// TIA Portal V20 export
FUNCTION_BLOCK "Sequence_1_TransferPnPLeft"   // FB32856, LAD
TITLE = Sequence
// Sequence template programmend in ladder logic
// stored: IsIECCheckEnabled true, MemoryReserve 100, Namespace Unit1.Em5, SetENOAutomatically true
   VAR_INPUT
      unitStatus { ExternalAccessible := 'False'; ExternalVisible := 'False'; ExternalWritable := 'False'} : "LAF_typeUnitStatus";
   END_VAR
   VAR
      instSequenceLADControl { ExternalAccessible := 'False'; ExternalVisible := 'False'; ExternalWritable := 'False'} : "LAF_ControlLadSequence";
      instSequenceLADStatus { ExternalAccessible := 'False'; ExternalVisible := 'False'; ExternalWritable := 'False'} : "LAF_StatusLadSequence";
      statTonTime { ExternalAccessible := 'False'; ExternalVisible := 'False'; ExternalWritable := 'False'} : Array[0..9999] of TON_TIME;
      NoDataCheck { S7_SetPoint := 'True'} : "LER_typePartData";
   END_VAR
   VAR_TEMP
      tempCustomerAction : Bool;   // Placeholder for possible actions
      tempDo_nothing_and_wait_for_init : Bool;   // Placeholder for doing nothing
      tempSafeStateCondition : Bool;   // Temp Condition for the equipment module to be in a safe state
   END_VAR
   VAR CONSTANT
      delayTime : Time := T#500ms;
      STEP_IDLE : DInt := 1;
      JOB_1_STEP_01 : DInt := 101;
      JOB_1_STEP_10 : DInt := 110;
      JOB_1_STEP_20 : DInt := 120;
      JOB_1_STEP_30 : DInt := 130;
      JOB_1_STEP_40 : DInt := 140;
      JOB_1_STEP_50 : DInt := 150;
      JOB_1_STEP_60 : DInt := 160;
      JOB_1_STEP_70 : DInt := 170;
      JOB_1_STEP_80 : DInt := 180;
      JOB_1_STEP_90 : DInt := 190;
      JOB_2_STEP_01 : DInt := 201;
      JOB_2_STEP_10 : DInt := 210;
      JOB_2_STEP_20 : DInt := 220;
      JOB_2_STEP_30 : DInt := 230;
      JOB_2_STEP_40 : DInt := 240;
      JOB_2_STEP_41 : DInt := 241;
      JOB_2_STEP_42 : DInt := 242;
      JOB_2_STEP_50 : DInt := 250;
      JOB_2_STEP_80 : DInt := 280;
      JOB_2_STEP_81 : DInt := 281;
      JOB_2_STEP_90 : DInt := 290;
      JOB_3_STEP_01 : DInt := 301;
      JOB_3_STEP_10 : DInt := 310;
      JOB_3_STEP_20 : DInt := 320;
      JOB_3_STEP_30 : DInt := 330;
      JOB_3_STEP_40 : DInt := 340;
      JOB_3_STEP_50 : DInt := 350;
      JOB_3_STEP_51 : DInt := 351;
      JOB_3_STEP_80 : DInt := 380;
      JOB_3_STEP_81 : DInt := 381;
      JOB_3_STEP_90 : DInt := 390;
      JOB_4_STEP_01 : DInt := 401;
      JOB_4_STEP_10 : DInt := 410;
      JOB_4_STEP_20 : DInt := 420;
      JOB_4_STEP_30 : DInt := 430;
      JOB_4_STEP_40 : DInt := 440;
      JOB_4_STEP_41 : DInt := 441;
      JOB_4_STEP_80 : DInt := 480;
      JOB_4_STEP_81 : DInt := 481;
      JOB_4_STEP_90 : DInt := 490;
      JOB_5_STEP_01 : DInt := 501;
      JOB_5_STEP_10 : DInt := 510;
      JOB_5_STEP_20 : DInt := 520;
      JOB_5_STEP_30 : DInt := 530;
      JOB_5_STEP_40 : DInt := 540;
      JOB_5_STEP_41 : DInt := 541;
      JOB_5_STEP_42 : DInt := 542;
      JOB_5_STEP_80 : DInt := 580;
      JOB_5_STEP_81 : DInt := 581;
      JOB_5_STEP_90 : DInt := 590;
      JOB_6_STEP_01 : DInt := 601;
      JOB_6_STEP_10 : DInt := 610;
      JOB_6_STEP_20 : DInt := 620;
      JOB_6_STEP_30 : DInt := 630;
      JOB_6_STEP_40 : DInt := 640;
      JOB_6_STEP_50 : DInt := 650;
      JOB_6_STEP_51 : DInt := 651;
      JOB_6_STEP_80 : DInt := 680;
      JOB_6_STEP_81 : DInt := 681;
      JOB_6_STEP_90 : DInt := 690;
      JOB_7_STEP_01 : DInt := 701;
      JOB_7_STEP_10 : DInt := 710;
      JOB_7_STEP_20 : DInt := 720;
      JOB_7_STEP_30 : DInt := 730;
      JOB_7_STEP_40 : DInt := 740;
      JOB_7_STEP_41 : DInt := 741;
      JOB_7_STEP_80 : DInt := 780;
      JOB_7_STEP_81 : DInt := 781;
      JOB_7_STEP_90 : DInt := 790;
      JOB_9_STEP_01 : DInt := 901;
      JOB_9_STEP_10 : DInt := 910;
      JOB_9_STEP_20 : DInt := 920;
      JOB_9_STEP_30 : DInt := 930;
      JOB_9_STEP_40 : DInt := 940;
      JOB_9_STEP_50 : DInt := 950;
      JOB_9_STEP_51 : DInt := 951;
      JOB_9_STEP_80 : DInt := 980;
      JOB_9_STEP_81 : DInt := 981;
      JOB_9_STEP_82 : DInt := 982;
      JOB_9_STEP_90 : DInt := 990;
      STEP_IMMEDIATE_STOP : DInt := 9001;   // Step executed when an immediate stop command is triggered for the sequence (i.e. when unit is in state aborting)
   END_VAR
   VAR_TEMP   // added for the SCL form of the ladder/FBD networks
      _w1 : Bool;
      _w2 : Bool;
      _w3 : Bool;
      _w4 : Bool;
      _w5 : Bool;
      _w6 : Bool;
      _w7 : Bool;
   END_VAR
BEGIN

REGION Network 1: BLOCK INFO HEADER
   // (company) / (C) Copyright (year)
   // ---------------------------------------------------------------------------------
   // Title:                             (Title of this block)
   // Comment/Function: (that is implemented in the block)
   // Library/Family:           (that the source is dedicated to)
   // Author:                        (department / person in charge / contact)
   // Target System:          (test system with FW version)
   // Engineering:              TIA Portal (SW version)
   // Restrictions:               (OB types, etc.)
   // Requirements:           (hardware, technological package, etc.)
   // ---------------------------------------------------------------------------------
   // Change log table:
   // Version          | Date             | Signature      | Expert in charge  | Changes applied ------------------------|----------------------|-------------------------|--------------------------------|-----------------------
   // 001.000.000 | yyyy-mm-dd | 0x00000000 | (name of expert) | First released version
END_REGION

REGION Network 2: DESCRIPTION
   // This is a template block provided by the Automation Framework. It can be used to create an own project.
   // The Block Info Header is prepared to put in your own data.
   // Description of the block could be added here and the docu created by Code2Docu.
END_REGION

REGION Network 3: ********************* CONTROL *************************
END_REGION

REGION Network 4: Sequence Control ("Enter your Sequins number here")
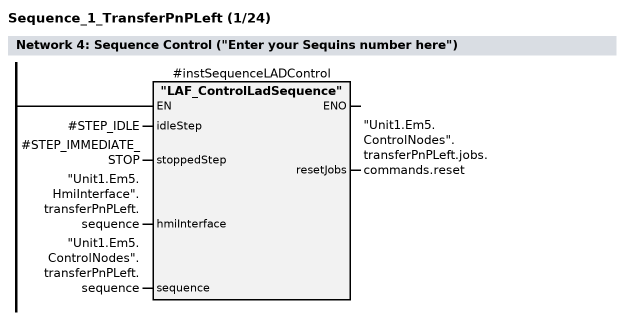
   RUNG wire#powerrail
      #instSequenceLADControl(idleStep := #STEP_IDLE, stoppedStep := #STEP_IMMEDIATE_STOP, hmiInterface := "Unit1.Em5.HmiInterface".transferPnPLeft.sequence, sequence := "Unit1.Em5.ControlNodes".transferPnPLeft.sequence, resetJobs => "Unit1.Em5.ControlNodes".transferPnPLeft.jobs.commands.reset)
   END_RUNG
   // the same network as SCL:
   #instSequenceLADControl(idleStep := #STEP_IDLE,   // "LAF_ControlLadSequence"
                           stoppedStep := #STEP_IMMEDIATE_STOP,
                           hmiInterface := "Unit1.Em5.HmiInterface".transferPnPLeft.sequence,
                           sequence := "Unit1.Em5.ControlNodes".transferPnPLeft.sequence,
                           resetJobs => "Unit1.Em5.ControlNodes".transferPnPLeft.jobs.commands.reset);
END_REGION

REGION Network 5: Step IDLE
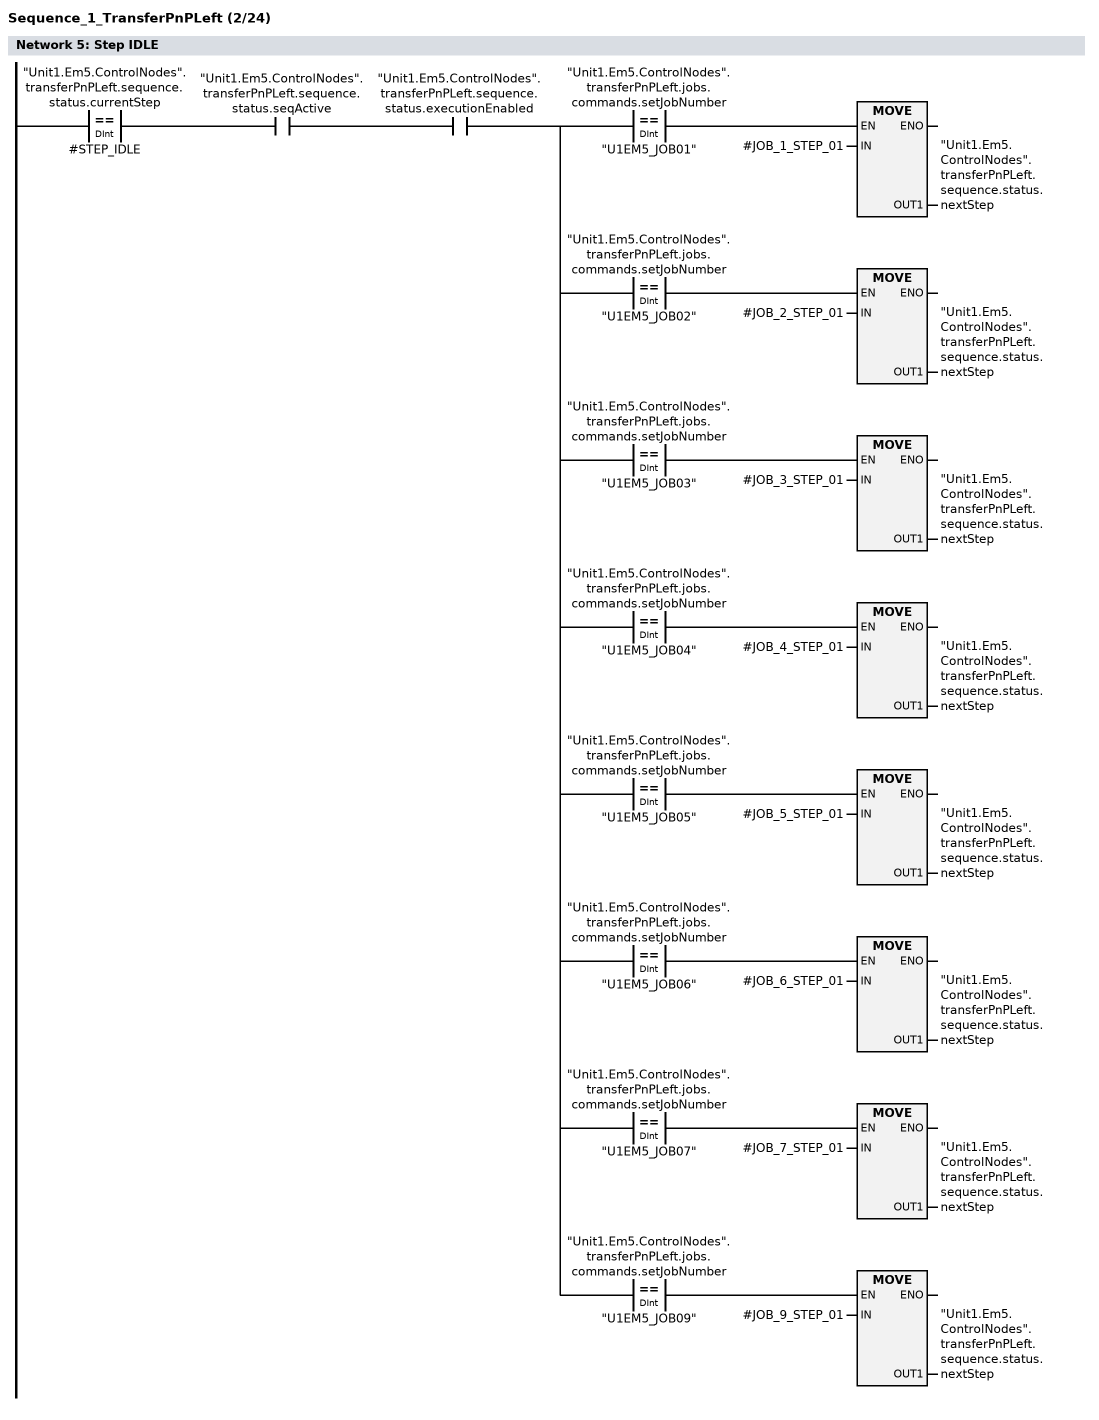
   RUNG wire#powerrail
      { S7_Templates := "SrcType := DInt" } EQ_Contact(in1 := "Unit1.Em5.ControlNodes".transferPnPLeft.sequence.status.currentStep, in2 := #STEP_IDLE)
      Contact( "Unit1.Em5.ControlNodes".transferPnPLeft.sequence.status.seqActive )
      Contact( "Unit1.Em5.ControlNodes".transferPnPLeft.sequence.status.executionEnabled )
      wire#w1
      { S7_Templates := "SrcType := DInt" } EQ_Contact(in1 := "Unit1.Em5.ControlNodes".transferPnPLeft.jobs.commands.setJobNumber, in2 := "U1EM5_JOB01")
      Move(in := #JOB_1_STEP_01, out1 => "Unit1.Em5.ControlNodes".transferPnPLeft.sequence.status.nextStep)
   END_RUNG
   RUNG wire#w1
      { S7_Templates := "SrcType := DInt" } EQ_Contact(in1 := "Unit1.Em5.ControlNodes".transferPnPLeft.jobs.commands.setJobNumber, in2 := "U1EM5_JOB02")
      Move(in := #JOB_2_STEP_01, out1 => "Unit1.Em5.ControlNodes".transferPnPLeft.sequence.status.nextStep)
   END_RUNG
   RUNG wire#w1
      { S7_Templates := "SrcType := DInt" } EQ_Contact(in1 := "Unit1.Em5.ControlNodes".transferPnPLeft.jobs.commands.setJobNumber, in2 := "U1EM5_JOB03")
      Move(in := #JOB_3_STEP_01, out1 => "Unit1.Em5.ControlNodes".transferPnPLeft.sequence.status.nextStep)
   END_RUNG
   RUNG wire#w1
      { S7_Templates := "SrcType := DInt" } EQ_Contact(in1 := "Unit1.Em5.ControlNodes".transferPnPLeft.jobs.commands.setJobNumber, in2 := "U1EM5_JOB04")
      Move(in := #JOB_4_STEP_01, out1 => "Unit1.Em5.ControlNodes".transferPnPLeft.sequence.status.nextStep)
   END_RUNG
   RUNG wire#w1
      { S7_Templates := "SrcType := DInt" } EQ_Contact(in1 := "Unit1.Em5.ControlNodes".transferPnPLeft.jobs.commands.setJobNumber, in2 := "U1EM5_JOB05")
      Move(in := #JOB_5_STEP_01, out1 => "Unit1.Em5.ControlNodes".transferPnPLeft.sequence.status.nextStep)
   END_RUNG
   RUNG wire#w1
      { S7_Templates := "SrcType := DInt" } EQ_Contact(in1 := "Unit1.Em5.ControlNodes".transferPnPLeft.jobs.commands.setJobNumber, in2 := "U1EM5_JOB06")
      Move(in := #JOB_6_STEP_01, out1 => "Unit1.Em5.ControlNodes".transferPnPLeft.sequence.status.nextStep)
   END_RUNG
   RUNG wire#w1
      { S7_Templates := "SrcType := DInt" } EQ_Contact(in1 := "Unit1.Em5.ControlNodes".transferPnPLeft.jobs.commands.setJobNumber, in2 := "U1EM5_JOB07")
      Move(in := #JOB_7_STEP_01, out1 => "Unit1.Em5.ControlNodes".transferPnPLeft.sequence.status.nextStep)
   END_RUNG
   RUNG wire#w1
      { S7_Templates := "SrcType := DInt" } EQ_Contact(in1 := "Unit1.Em5.ControlNodes".transferPnPLeft.jobs.commands.setJobNumber, in2 := "U1EM5_JOB09")
      Move(in := #JOB_9_STEP_01, out1 => "Unit1.Em5.ControlNodes".transferPnPLeft.sequence.status.nextStep)
   END_RUNG
   // the same network as SCL:
   #_w1 := ("Unit1.Em5.ControlNodes".transferPnPLeft.sequence.status.currentStep = #STEP_IDLE) AND "Unit1.Em5.ControlNodes".transferPnPLeft.sequence.status.seqActive AND "Unit1.Em5.ControlNodes".transferPnPLeft.sequence.status.executionEnabled;
   IF #_w1 AND ("Unit1.Em5.ControlNodes".transferPnPLeft.jobs.commands.setJobNumber = "U1EM5_JOB01") THEN
       "Unit1.Em5.ControlNodes".transferPnPLeft.sequence.status.nextStep := #JOB_1_STEP_01;
   END_IF;
   IF #_w1 AND ("Unit1.Em5.ControlNodes".transferPnPLeft.jobs.commands.setJobNumber = "U1EM5_JOB02") THEN
       "Unit1.Em5.ControlNodes".transferPnPLeft.sequence.status.nextStep := #JOB_2_STEP_01;
   END_IF;
   IF #_w1 AND ("Unit1.Em5.ControlNodes".transferPnPLeft.jobs.commands.setJobNumber = "U1EM5_JOB03") THEN
       "Unit1.Em5.ControlNodes".transferPnPLeft.sequence.status.nextStep := #JOB_3_STEP_01;
   END_IF;
   IF #_w1 AND ("Unit1.Em5.ControlNodes".transferPnPLeft.jobs.commands.setJobNumber = "U1EM5_JOB04") THEN
       "Unit1.Em5.ControlNodes".transferPnPLeft.sequence.status.nextStep := #JOB_4_STEP_01;
   END_IF;
   IF #_w1 AND ("Unit1.Em5.ControlNodes".transferPnPLeft.jobs.commands.setJobNumber = "U1EM5_JOB05") THEN
       "Unit1.Em5.ControlNodes".transferPnPLeft.sequence.status.nextStep := #JOB_5_STEP_01;
   END_IF;
   IF #_w1 AND ("Unit1.Em5.ControlNodes".transferPnPLeft.jobs.commands.setJobNumber = "U1EM5_JOB06") THEN
       "Unit1.Em5.ControlNodes".transferPnPLeft.sequence.status.nextStep := #JOB_6_STEP_01;
   END_IF;
   IF #_w1 AND ("Unit1.Em5.ControlNodes".transferPnPLeft.jobs.commands.setJobNumber = "U1EM5_JOB07") THEN
       "Unit1.Em5.ControlNodes".transferPnPLeft.sequence.status.nextStep := #JOB_7_STEP_01;
   END_IF;
   IF #_w1 AND ("Unit1.Em5.ControlNodes".transferPnPLeft.jobs.commands.setJobNumber = "U1EM5_JOB09") THEN
       "Unit1.Em5.ControlNodes".transferPnPLeft.sequence.status.nextStep := #JOB_9_STEP_01;
   END_IF;
END_REGION

REGION Network 6: *************** JOB[1] EM HOMING ************************
END_REGION

REGION Network 7: Step[101] : JOB[1] Condition
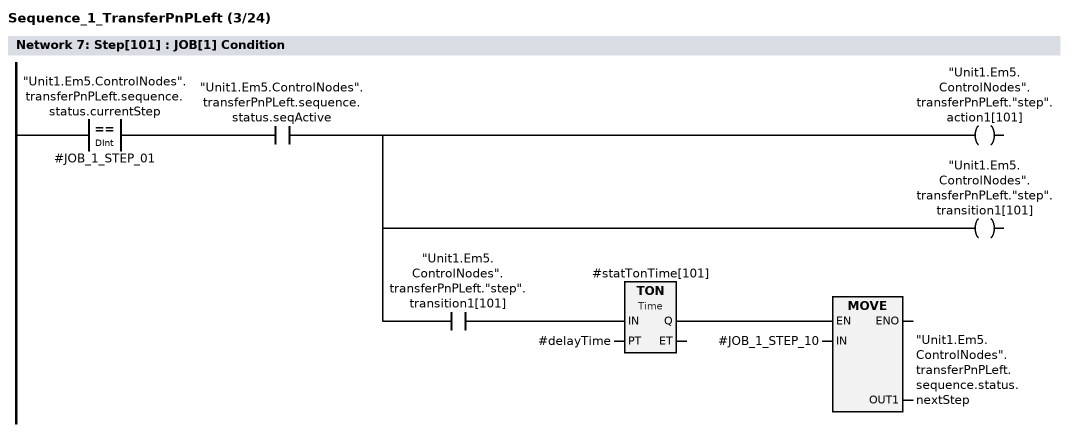
   RUNG wire#powerrail
      { S7_Templates := "SrcType := DInt" } EQ_Contact(in1 := "Unit1.Em5.ControlNodes".transferPnPLeft.sequence.status.currentStep, in2 := #JOB_1_STEP_01)
      Contact( "Unit1.Em5.ControlNodes".transferPnPLeft.sequence.status.seqActive )
      wire#w1
      Coil( "Unit1.Em5.ControlNodes".transferPnPLeft."step".action1[101] )
   END_RUNG
   RUNG wire#w1
      Coil( "Unit1.Em5.ControlNodes".transferPnPLeft."step".transition1[101] )
   END_RUNG
   RUNG wire#w1
      Contact( "Unit1.Em5.ControlNodes".transferPnPLeft."step".transition1[101] )
      { S7_Templates := "time_type := Time" } #statTonTime[101].TON(pt := #delayTime, et =>)
      Move(in := #JOB_1_STEP_10, out1 => "Unit1.Em5.ControlNodes".transferPnPLeft.sequence.status.nextStep)
   END_RUNG
   // the same network as SCL:
   "Unit1.Em5.ControlNodes".transferPnPLeft."step".action1[101] := ("Unit1.Em5.ControlNodes".transferPnPLeft.sequence.status.currentStep = #JOB_1_STEP_01) AND "Unit1.Em5.ControlNodes".transferPnPLeft.sequence.status.seqActive;
   "Unit1.Em5.ControlNodes".transferPnPLeft."step".transition1[101] := ("Unit1.Em5.ControlNodes".transferPnPLeft.sequence.status.currentStep = #JOB_1_STEP_01) AND "Unit1.Em5.ControlNodes".transferPnPLeft.sequence.status.seqActive;
   #statTonTime[101].TON(IN := ("Unit1.Em5.ControlNodes".transferPnPLeft.sequence.status.currentStep = #JOB_1_STEP_01) AND "Unit1.Em5.ControlNodes".transferPnPLeft.sequence.status.seqActive AND "Unit1.Em5.ControlNodes".transferPnPLeft."step".transition1[101],
                         PT := #delayTime);
   IF #statTonTime[101].Q THEN
       "Unit1.Em5.ControlNodes".transferPnPLeft.sequence.status.nextStep := #JOB_1_STEP_10;
   END_IF;
END_REGION

REGION Network 8: Step[110] : Transfer PP Left Clamp Open
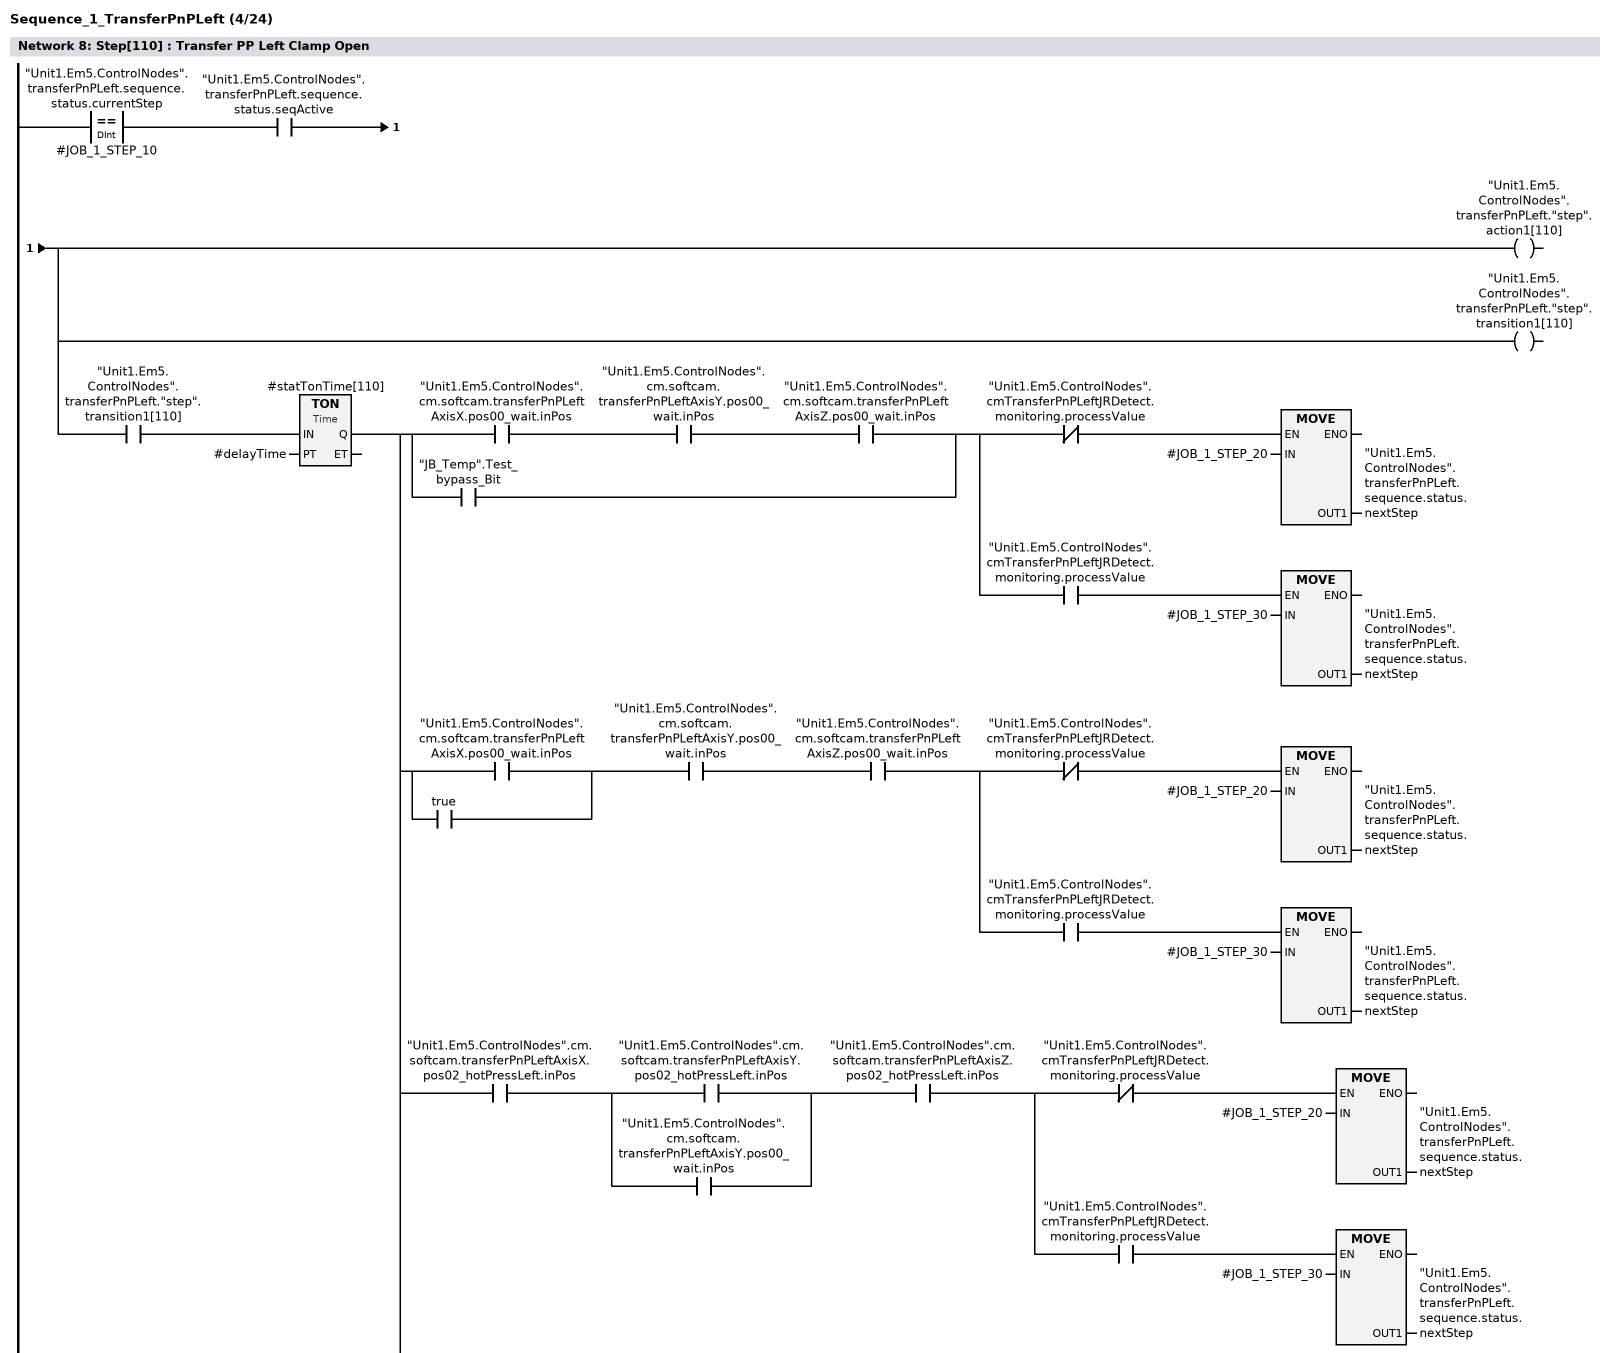
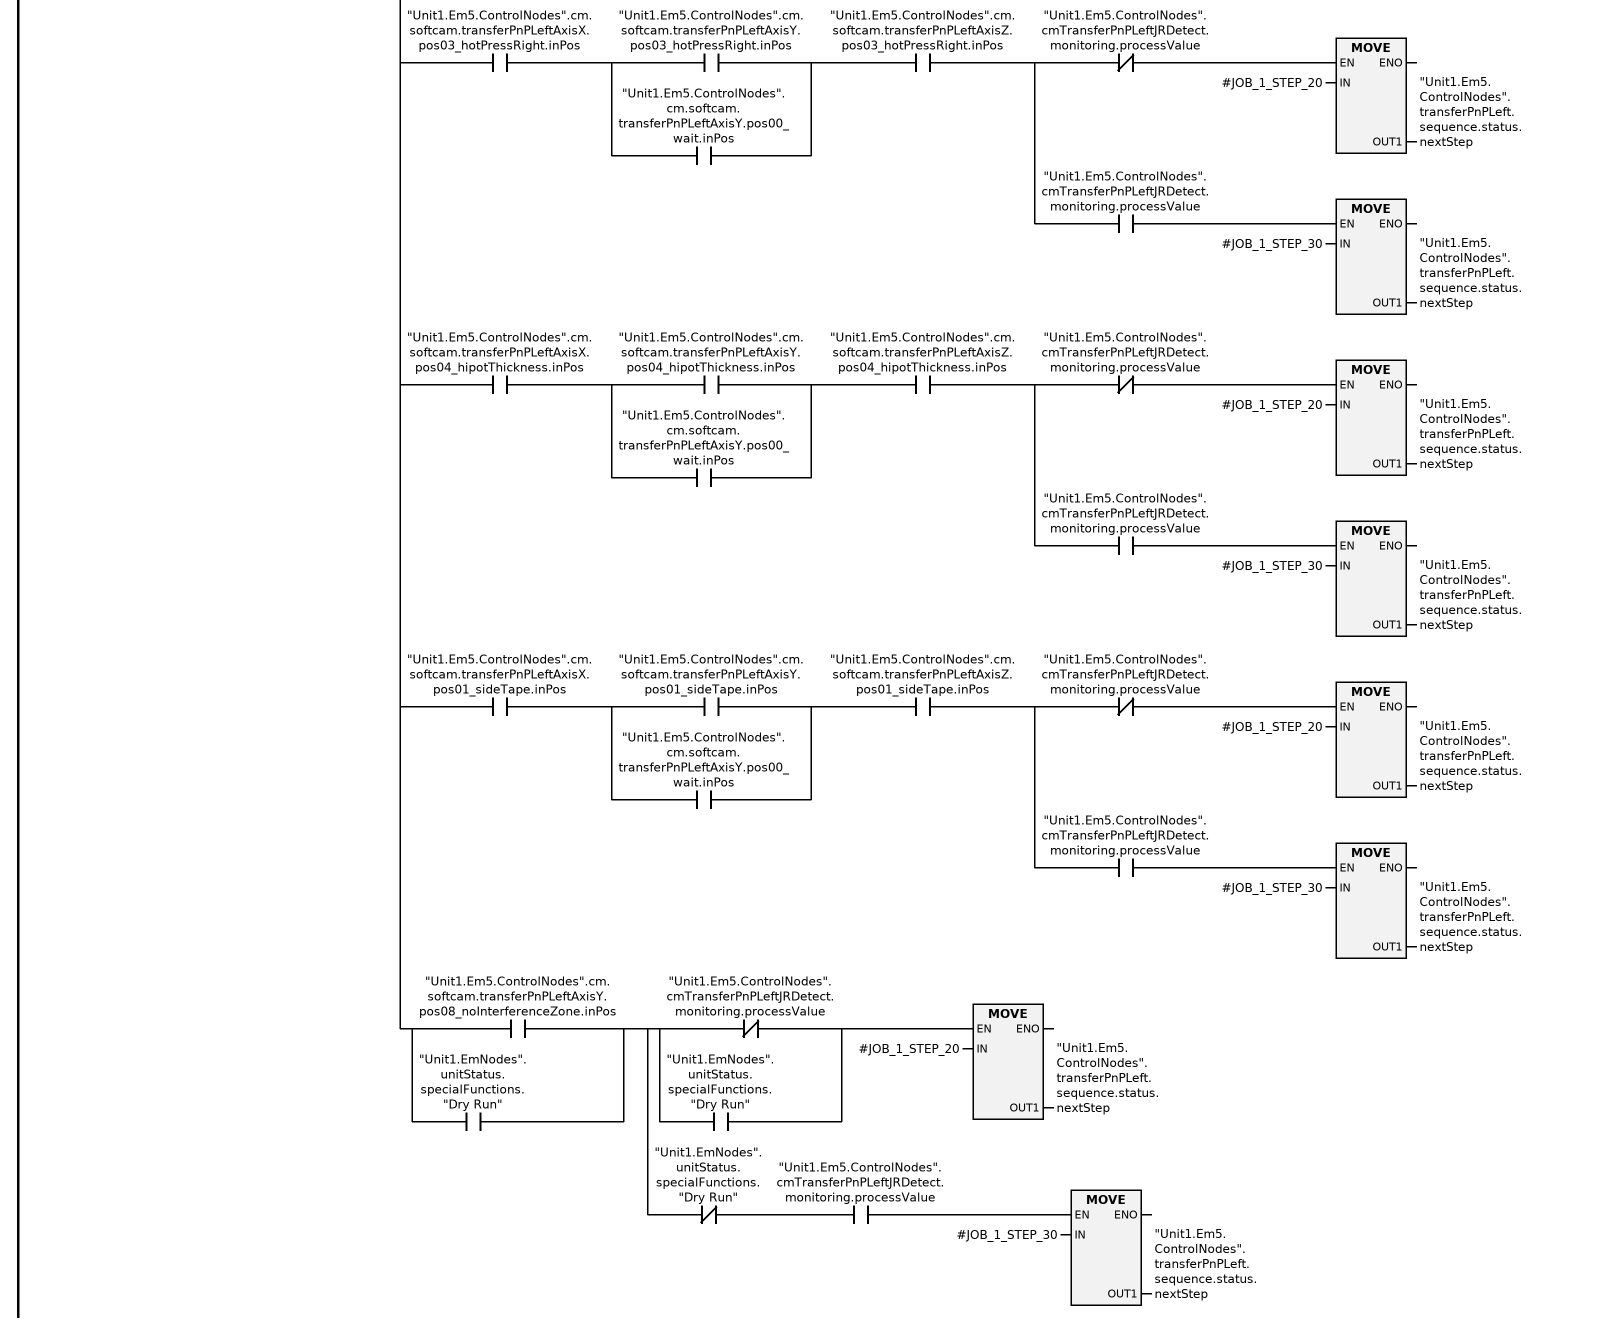
   RUNG wire#powerrail
      { S7_Templates := "SrcType := DInt" } EQ_Contact(in1 := "Unit1.Em5.ControlNodes".transferPnPLeft.sequence.status.currentStep, in2 := #JOB_1_STEP_10)
      Contact( "Unit1.Em5.ControlNodes".transferPnPLeft.sequence.status.seqActive )
      wire#w1
      Coil( "Unit1.Em5.ControlNodes".transferPnPLeft."step".action1[110] )
   END_RUNG
   RUNG wire#w1
      Coil( "Unit1.Em5.ControlNodes".transferPnPLeft."step".transition1[110] )
   END_RUNG
   RUNG wire#w1
      Contact( "Unit1.Em5.ControlNodes".transferPnPLeft."step".transition1[110] )
      { S7_Templates := "time_type := Time" } #statTonTime[110].TON(pt := #delayTime, et =>)
      wire#w2
      Contact( "Unit1.Em5.ControlNodes".cm.softcam.transferPnPLeftAxisX.pos00_wait.inPos )
      Contact( "Unit1.Em5.ControlNodes".cm.softcam.transferPnPLeftAxisY.pos00_wait.inPos )
      Contact( "Unit1.Em5.ControlNodes".cm.softcam.transferPnPLeftAxisZ.pos00_wait.inPos )
      wire#w3
      I_Contact( "Unit1.Em5.ControlNodes".cmTransferPnPLeftJRDetect.monitoring.processValue )
      Move(in := #JOB_1_STEP_20, out1 => "Unit1.Em5.ControlNodes".transferPnPLeft.sequence.status.nextStep)
   END_RUNG
   RUNG wire#w2
      Contact( "JB_Temp".Test_bypass_Bit )
   END_RUNG wire#w3
   RUNG wire#w3
      Contact( "Unit1.Em5.ControlNodes".cmTransferPnPLeftJRDetect.monitoring.processValue )
      Move(in := #JOB_1_STEP_30, out1 => "Unit1.Em5.ControlNodes".transferPnPLeft.sequence.status.nextStep)
   END_RUNG
   RUNG wire#w2
      Contact( "Unit1.Em5.ControlNodes".cm.softcam.transferPnPLeftAxisX.pos00_wait.inPos )
      wire#w4
      Contact( "Unit1.Em5.ControlNodes".cm.softcam.transferPnPLeftAxisY.pos00_wait.inPos )
      Contact( "Unit1.Em5.ControlNodes".cm.softcam.transferPnPLeftAxisZ.pos00_wait.inPos )
      wire#w5
      I_Contact( "Unit1.Em5.ControlNodes".cmTransferPnPLeftJRDetect.monitoring.processValue )
      Move(in := #JOB_1_STEP_20, out1 => "Unit1.Em5.ControlNodes".transferPnPLeft.sequence.status.nextStep)
   END_RUNG
   RUNG wire#w2
      Contact( true )
   END_RUNG wire#w4
   RUNG wire#w5
      Contact( "Unit1.Em5.ControlNodes".cmTransferPnPLeftJRDetect.monitoring.processValue )
      Move(in := #JOB_1_STEP_30, out1 => "Unit1.Em5.ControlNodes".transferPnPLeft.sequence.status.nextStep)
   END_RUNG
   RUNG wire#w2
      Contact( "Unit1.Em5.ControlNodes".cm.softcam.transferPnPLeftAxisX.pos02_hotPressLeft.inPos )
      wire#w6
      Contact( "Unit1.Em5.ControlNodes".cm.softcam.transferPnPLeftAxisY.pos02_hotPressLeft.inPos )
      wire#w7
      Contact( "Unit1.Em5.ControlNodes".cm.softcam.transferPnPLeftAxisZ.pos02_hotPressLeft.inPos )
      wire#w8
      I_Contact( "Unit1.Em5.ControlNodes".cmTransferPnPLeftJRDetect.monitoring.processValue )
      Move(in := #JOB_1_STEP_20, out1 => "Unit1.Em5.ControlNodes".transferPnPLeft.sequence.status.nextStep)
   END_RUNG
   RUNG wire#w6
      Contact( "Unit1.Em5.ControlNodes".cm.softcam.transferPnPLeftAxisY.pos00_wait.inPos )
   END_RUNG wire#w7
   RUNG wire#w8
      Contact( "Unit1.Em5.ControlNodes".cmTransferPnPLeftJRDetect.monitoring.processValue )
      Move(in := #JOB_1_STEP_30, out1 => "Unit1.Em5.ControlNodes".transferPnPLeft.sequence.status.nextStep)
   END_RUNG
   RUNG wire#w2
      Contact( "Unit1.Em5.ControlNodes".cm.softcam.transferPnPLeftAxisX.pos03_hotPressRight.inPos )
      wire#w9
      Contact( "Unit1.Em5.ControlNodes".cm.softcam.transferPnPLeftAxisY.pos03_hotPressRight.inPos )
      wire#w10
      Contact( "Unit1.Em5.ControlNodes".cm.softcam.transferPnPLeftAxisZ.pos03_hotPressRight.inPos )
      wire#w11
      I_Contact( "Unit1.Em5.ControlNodes".cmTransferPnPLeftJRDetect.monitoring.processValue )
      Move(in := #JOB_1_STEP_20, out1 => "Unit1.Em5.ControlNodes".transferPnPLeft.sequence.status.nextStep)
   END_RUNG
   RUNG wire#w9
      Contact( "Unit1.Em5.ControlNodes".cm.softcam.transferPnPLeftAxisY.pos00_wait.inPos )
   END_RUNG wire#w10
   RUNG wire#w11
      Contact( "Unit1.Em5.ControlNodes".cmTransferPnPLeftJRDetect.monitoring.processValue )
      Move(in := #JOB_1_STEP_30, out1 => "Unit1.Em5.ControlNodes".transferPnPLeft.sequence.status.nextStep)
   END_RUNG
   RUNG wire#w2
      Contact( "Unit1.Em5.ControlNodes".cm.softcam.transferPnPLeftAxisX.pos04_hipotThickness.inPos )
      wire#w12
      Contact( "Unit1.Em5.ControlNodes".cm.softcam.transferPnPLeftAxisY.pos04_hipotThickness.inPos )
      wire#w13
      Contact( "Unit1.Em5.ControlNodes".cm.softcam.transferPnPLeftAxisZ.pos04_hipotThickness.inPos )
      wire#w14
      I_Contact( "Unit1.Em5.ControlNodes".cmTransferPnPLeftJRDetect.monitoring.processValue )
      Move(in := #JOB_1_STEP_20, out1 => "Unit1.Em5.ControlNodes".transferPnPLeft.sequence.status.nextStep)
   END_RUNG
   RUNG wire#w12
      Contact( "Unit1.Em5.ControlNodes".cm.softcam.transferPnPLeftAxisY.pos00_wait.inPos )
   END_RUNG wire#w13
   RUNG wire#w14
      Contact( "Unit1.Em5.ControlNodes".cmTransferPnPLeftJRDetect.monitoring.processValue )
      Move(in := #JOB_1_STEP_30, out1 => "Unit1.Em5.ControlNodes".transferPnPLeft.sequence.status.nextStep)
   END_RUNG
   RUNG wire#w2
      Contact( "Unit1.Em5.ControlNodes".cm.softcam.transferPnPLeftAxisX.pos01_sideTape.inPos )
      wire#w15
      Contact( "Unit1.Em5.ControlNodes".cm.softcam.transferPnPLeftAxisY.pos01_sideTape.inPos )
      wire#w16
      Contact( "Unit1.Em5.ControlNodes".cm.softcam.transferPnPLeftAxisZ.pos01_sideTape.inPos )
      wire#w17
      I_Contact( "Unit1.Em5.ControlNodes".cmTransferPnPLeftJRDetect.monitoring.processValue )
      Move(in := #JOB_1_STEP_20, out1 => "Unit1.Em5.ControlNodes".transferPnPLeft.sequence.status.nextStep)
   END_RUNG
   RUNG wire#w15
      Contact( "Unit1.Em5.ControlNodes".cm.softcam.transferPnPLeftAxisY.pos00_wait.inPos )
   END_RUNG wire#w16
   RUNG wire#w17
      Contact( "Unit1.Em5.ControlNodes".cmTransferPnPLeftJRDetect.monitoring.processValue )
      Move(in := #JOB_1_STEP_30, out1 => "Unit1.Em5.ControlNodes".transferPnPLeft.sequence.status.nextStep)
   END_RUNG
   RUNG wire#w2
      Contact( "Unit1.Em5.ControlNodes".cm.softcam.transferPnPLeftAxisY.pos08_noInterferenceZone.inPos )
      wire#w18
      I_Contact( "Unit1.Em5.ControlNodes".cmTransferPnPLeftJRDetect.monitoring.processValue )
      wire#w19
      Move(in := #JOB_1_STEP_20, out1 => "Unit1.Em5.ControlNodes".transferPnPLeft.sequence.status.nextStep)
   END_RUNG
   RUNG wire#w2
      Contact( "Unit1.EmNodes".unitStatus.specialFunctions."Dry Run" )
   END_RUNG wire#w18
   RUNG wire#w18
      Contact( "Unit1.EmNodes".unitStatus.specialFunctions."Dry Run" )
   END_RUNG wire#w19
   RUNG wire#w18
      I_Contact( "Unit1.EmNodes".unitStatus.specialFunctions."Dry Run" )
      Contact( "Unit1.Em5.ControlNodes".cmTransferPnPLeftJRDetect.monitoring.processValue )
      Move(in := #JOB_1_STEP_30, out1 => "Unit1.Em5.ControlNodes".transferPnPLeft.sequence.status.nextStep)
   END_RUNG
   // the same network as SCL:
   "Unit1.Em5.ControlNodes".transferPnPLeft."step".action1[110] := ("Unit1.Em5.ControlNodes".transferPnPLeft.sequence.status.currentStep = #JOB_1_STEP_10) AND "Unit1.Em5.ControlNodes".transferPnPLeft.sequence.status.seqActive;
   "Unit1.Em5.ControlNodes".transferPnPLeft."step".transition1[110] := ("Unit1.Em5.ControlNodes".transferPnPLeft.sequence.status.currentStep = #JOB_1_STEP_10) AND "Unit1.Em5.ControlNodes".transferPnPLeft.sequence.status.seqActive;
   #statTonTime[110].TON(IN := ("Unit1.Em5.ControlNodes".transferPnPLeft.sequence.status.currentStep = #JOB_1_STEP_10) AND "Unit1.Em5.ControlNodes".transferPnPLeft.sequence.status.seqActive AND "Unit1.Em5.ControlNodes".transferPnPLeft."step".transition1[110],
                         PT := #delayTime);
   #_w1 := #statTonTime[110].Q AND (("Unit1.Em5.ControlNodes".cm.softcam.transferPnPLeftAxisX.pos00_wait.inPos AND "Unit1.Em5.ControlNodes".cm.softcam.transferPnPLeftAxisY.pos00_wait.inPos AND "Unit1.Em5.ControlNodes".cm.softcam.transferPnPLeftAxisZ.pos00_wait.inPos) OR "JB_Temp".Test_bypass_Bit);
   IF #_w1 AND NOT "Unit1.Em5.ControlNodes".cmTransferPnPLeftJRDetect.monitoring.processValue THEN
       "Unit1.Em5.ControlNodes".transferPnPLeft.sequence.status.nextStep := #JOB_1_STEP_20;
   END_IF;
   IF #_w1 AND "Unit1.Em5.ControlNodes".cmTransferPnPLeftJRDetect.monitoring.processValue THEN
       "Unit1.Em5.ControlNodes".transferPnPLeft.sequence.status.nextStep := #JOB_1_STEP_30;
   END_IF;
   #_w2 := #statTonTime[110].Q AND ("Unit1.Em5.ControlNodes".cm.softcam.transferPnPLeftAxisX.pos00_wait.inPos OR true) AND "Unit1.Em5.ControlNodes".cm.softcam.transferPnPLeftAxisY.pos00_wait.inPos AND "Unit1.Em5.ControlNodes".cm.softcam.transferPnPLeftAxisZ.pos00_wait.inPos;
   IF #_w2 AND NOT "Unit1.Em5.ControlNodes".cmTransferPnPLeftJRDetect.monitoring.processValue THEN
       "Unit1.Em5.ControlNodes".transferPnPLeft.sequence.status.nextStep := #JOB_1_STEP_20;
   END_IF;
   IF #_w2 AND "Unit1.Em5.ControlNodes".cmTransferPnPLeftJRDetect.monitoring.processValue THEN
       "Unit1.Em5.ControlNodes".transferPnPLeft.sequence.status.nextStep := #JOB_1_STEP_30;
   END_IF;
   #_w3 := #statTonTime[110].Q AND "Unit1.Em5.ControlNodes".cm.softcam.transferPnPLeftAxisX.pos02_hotPressLeft.inPos AND ("Unit1.Em5.ControlNodes".cm.softcam.transferPnPLeftAxisY.pos02_hotPressLeft.inPos OR "Unit1.Em5.ControlNodes".cm.softcam.transferPnPLeftAxisY.pos00_wait.inPos) AND "Unit1.Em5.ControlNodes".cm.softcam.transferPnPLeftAxisZ.pos02_hotPressLeft.inPos;
   IF #_w3 AND NOT "Unit1.Em5.ControlNodes".cmTransferPnPLeftJRDetect.monitoring.processValue THEN
       "Unit1.Em5.ControlNodes".transferPnPLeft.sequence.status.nextStep := #JOB_1_STEP_20;
   END_IF;
   IF #_w3 AND "Unit1.Em5.ControlNodes".cmTransferPnPLeftJRDetect.monitoring.processValue THEN
       "Unit1.Em5.ControlNodes".transferPnPLeft.sequence.status.nextStep := #JOB_1_STEP_30;
   END_IF;
   #_w4 := #statTonTime[110].Q AND "Unit1.Em5.ControlNodes".cm.softcam.transferPnPLeftAxisX.pos03_hotPressRight.inPos AND ("Unit1.Em5.ControlNodes".cm.softcam.transferPnPLeftAxisY.pos03_hotPressRight.inPos OR "Unit1.Em5.ControlNodes".cm.softcam.transferPnPLeftAxisY.pos00_wait.inPos) AND "Unit1.Em5.ControlNodes".cm.softcam.transferPnPLeftAxisZ.pos03_hotPressRight.inPos;
   IF #_w4 AND NOT "Unit1.Em5.ControlNodes".cmTransferPnPLeftJRDetect.monitoring.processValue THEN
       "Unit1.Em5.ControlNodes".transferPnPLeft.sequence.status.nextStep := #JOB_1_STEP_20;
   END_IF;
   IF #_w4 AND "Unit1.Em5.ControlNodes".cmTransferPnPLeftJRDetect.monitoring.processValue THEN
       "Unit1.Em5.ControlNodes".transferPnPLeft.sequence.status.nextStep := #JOB_1_STEP_30;
   END_IF;
   #_w5 := #statTonTime[110].Q AND "Unit1.Em5.ControlNodes".cm.softcam.transferPnPLeftAxisX.pos04_hipotThickness.inPos AND ("Unit1.Em5.ControlNodes".cm.softcam.transferPnPLeftAxisY.pos04_hipotThickness.inPos OR "Unit1.Em5.ControlNodes".cm.softcam.transferPnPLeftAxisY.pos00_wait.inPos) AND "Unit1.Em5.ControlNodes".cm.softcam.transferPnPLeftAxisZ.pos04_hipotThickness.inPos;
   IF #_w5 AND NOT "Unit1.Em5.ControlNodes".cmTransferPnPLeftJRDetect.monitoring.processValue THEN
       "Unit1.Em5.ControlNodes".transferPnPLeft.sequence.status.nextStep := #JOB_1_STEP_20;
   END_IF;
   IF #_w5 AND "Unit1.Em5.ControlNodes".cmTransferPnPLeftJRDetect.monitoring.processValue THEN
       "Unit1.Em5.ControlNodes".transferPnPLeft.sequence.status.nextStep := #JOB_1_STEP_30;
   END_IF;
   #_w6 := #statTonTime[110].Q AND "Unit1.Em5.ControlNodes".cm.softcam.transferPnPLeftAxisX.pos01_sideTape.inPos AND ("Unit1.Em5.ControlNodes".cm.softcam.transferPnPLeftAxisY.pos01_sideTape.inPos OR "Unit1.Em5.ControlNodes".cm.softcam.transferPnPLeftAxisY.pos00_wait.inPos) AND "Unit1.Em5.ControlNodes".cm.softcam.transferPnPLeftAxisZ.pos01_sideTape.inPos;
   IF #_w6 AND NOT "Unit1.Em5.ControlNodes".cmTransferPnPLeftJRDetect.monitoring.processValue THEN
       "Unit1.Em5.ControlNodes".transferPnPLeft.sequence.status.nextStep := #JOB_1_STEP_20;
   END_IF;
   IF #_w6 AND "Unit1.Em5.ControlNodes".cmTransferPnPLeftJRDetect.monitoring.processValue THEN
       "Unit1.Em5.ControlNodes".transferPnPLeft.sequence.status.nextStep := #JOB_1_STEP_30;
   END_IF;
   #_w7 := #statTonTime[110].Q AND ("Unit1.Em5.ControlNodes".cm.softcam.transferPnPLeftAxisY.pos08_noInterferenceZone.inPos OR "Unit1.EmNodes".unitStatus.specialFunctions."Dry Run");
   IF #_w7 AND (NOT "Unit1.Em5.ControlNodes".cmTransferPnPLeftJRDetect.monitoring.processValue OR "Unit1.EmNodes".unitStatus.specialFunctions."Dry Run") THEN
       "Unit1.Em5.ControlNodes".transferPnPLeft.sequence.status.nextStep := #JOB_1_STEP_20;
   END_IF;
   IF #_w7 AND NOT "Unit1.EmNodes".unitStatus.specialFunctions."Dry Run" AND "Unit1.Em5.ControlNodes".cmTransferPnPLeftJRDetect.monitoring.processValue THEN
       "Unit1.Em5.ControlNodes".transferPnPLeft.sequence.status.nextStep := #JOB_1_STEP_30;
   END_IF;
END_REGION

REGION Network 9: Step[120] : Transfer PP Left Clamp Open
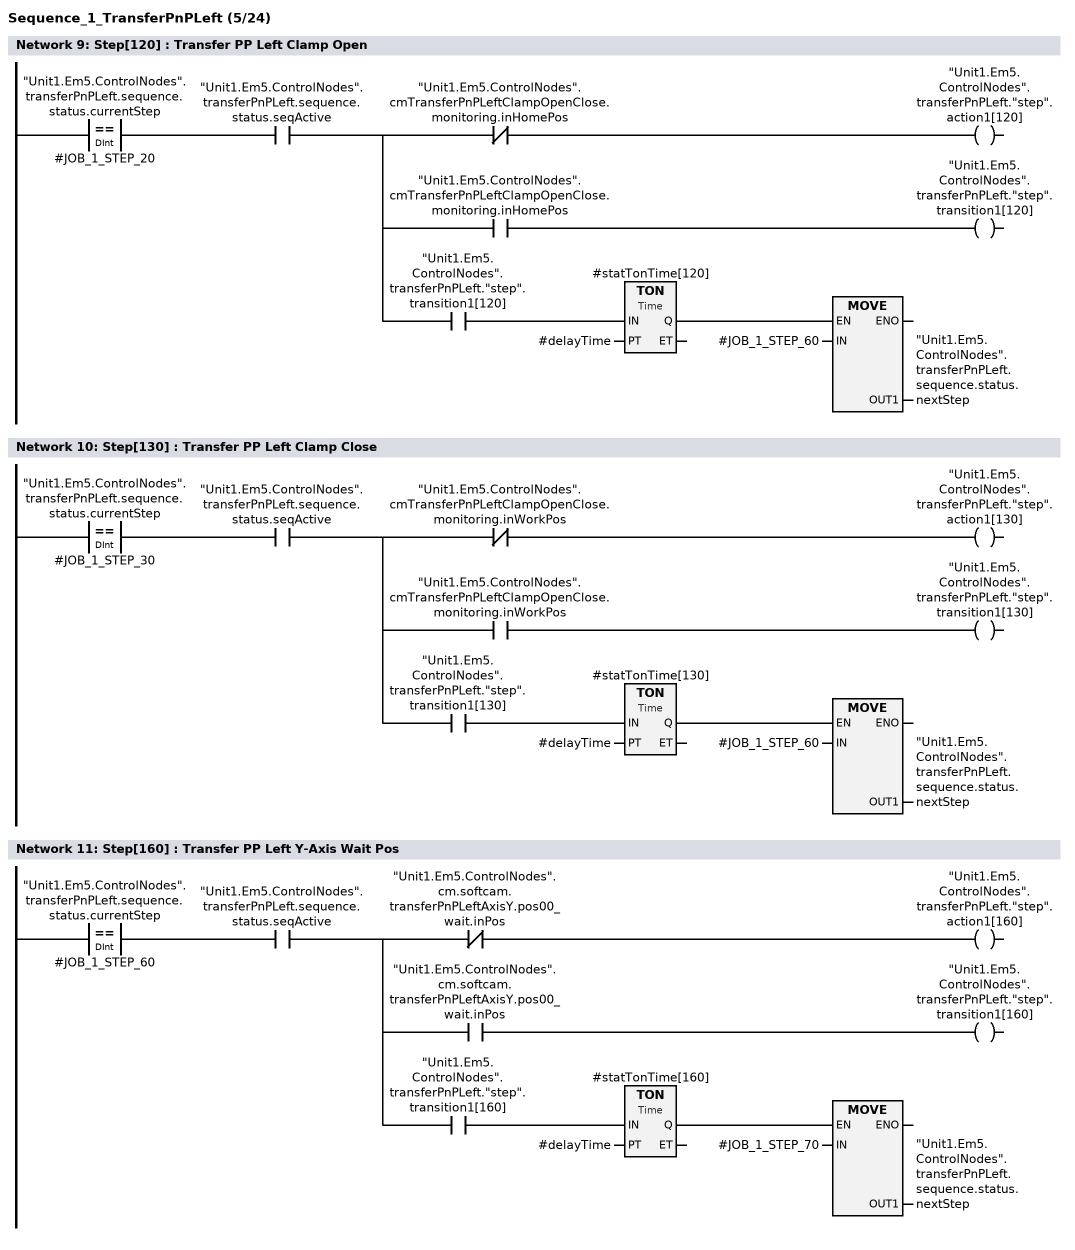
   RUNG wire#powerrail
      { S7_Templates := "SrcType := DInt" } EQ_Contact(in1 := "Unit1.Em5.ControlNodes".transferPnPLeft.sequence.status.currentStep, in2 := #JOB_1_STEP_20)
      Contact( "Unit1.Em5.ControlNodes".transferPnPLeft.sequence.status.seqActive )
      wire#w1
      I_Contact( "Unit1.Em5.ControlNodes".cmTransferPnPLeftClampOpenClose.monitoring.inHomePos )
      Coil( "Unit1.Em5.ControlNodes".transferPnPLeft."step".action1[120] )
   END_RUNG
   RUNG wire#w1
      Contact( "Unit1.Em5.ControlNodes".cmTransferPnPLeftClampOpenClose.monitoring.inHomePos )
      Coil( "Unit1.Em5.ControlNodes".transferPnPLeft."step".transition1[120] )
   END_RUNG
   RUNG wire#w1
      Contact( "Unit1.Em5.ControlNodes".transferPnPLeft."step".transition1[120] )
      { S7_Templates := "time_type := Time" } #statTonTime[120].TON(pt := #delayTime, et =>)
      Move(in := #JOB_1_STEP_60, out1 => "Unit1.Em5.ControlNodes".transferPnPLeft.sequence.status.nextStep)
   END_RUNG
   // the same network as SCL:
   #_w1 := ("Unit1.Em5.ControlNodes".transferPnPLeft.sequence.status.currentStep = #JOB_1_STEP_20) AND "Unit1.Em5.ControlNodes".transferPnPLeft.sequence.status.seqActive;
   "Unit1.Em5.ControlNodes".transferPnPLeft."step".action1[120] := #_w1 AND NOT "Unit1.Em5.ControlNodes".cmTransferPnPLeftClampOpenClose.monitoring.inHomePos;
   "Unit1.Em5.ControlNodes".transferPnPLeft."step".transition1[120] := #_w1 AND "Unit1.Em5.ControlNodes".cmTransferPnPLeftClampOpenClose.monitoring.inHomePos;
   #statTonTime[120].TON(IN := #_w1 AND "Unit1.Em5.ControlNodes".transferPnPLeft."step".transition1[120],
                         PT := #delayTime);
   IF #statTonTime[120].Q THEN
       "Unit1.Em5.ControlNodes".transferPnPLeft.sequence.status.nextStep := #JOB_1_STEP_60;
   END_IF;
END_REGION

REGION Network 10: Step[130] : Transfer PP Left Clamp Close
   RUNG wire#powerrail
      { S7_Templates := "SrcType := DInt" } EQ_Contact(in1 := "Unit1.Em5.ControlNodes".transferPnPLeft.sequence.status.currentStep, in2 := #JOB_1_STEP_30)
      Contact( "Unit1.Em5.ControlNodes".transferPnPLeft.sequence.status.seqActive )
      wire#w1
      I_Contact( "Unit1.Em5.ControlNodes".cmTransferPnPLeftClampOpenClose.monitoring.inWorkPos )
      Coil( "Unit1.Em5.ControlNodes".transferPnPLeft."step".action1[130] )
   END_RUNG
   RUNG wire#w1
      Contact( "Unit1.Em5.ControlNodes".cmTransferPnPLeftClampOpenClose.monitoring.inWorkPos )
      Coil( "Unit1.Em5.ControlNodes".transferPnPLeft."step".transition1[130] )
   END_RUNG
   RUNG wire#w1
      Contact( "Unit1.Em5.ControlNodes".transferPnPLeft."step".transition1[130] )
      { S7_Templates := "time_type := Time" } #statTonTime[130].TON(pt := #delayTime, et =>)
      Move(in := #JOB_1_STEP_60, out1 => "Unit1.Em5.ControlNodes".transferPnPLeft.sequence.status.nextStep)
   END_RUNG
   // the same network as SCL:
   #_w1 := ("Unit1.Em5.ControlNodes".transferPnPLeft.sequence.status.currentStep = #JOB_1_STEP_30) AND "Unit1.Em5.ControlNodes".transferPnPLeft.sequence.status.seqActive;
   "Unit1.Em5.ControlNodes".transferPnPLeft."step".action1[130] := #_w1 AND NOT "Unit1.Em5.ControlNodes".cmTransferPnPLeftClampOpenClose.monitoring.inWorkPos;
   "Unit1.Em5.ControlNodes".transferPnPLeft."step".transition1[130] := #_w1 AND "Unit1.Em5.ControlNodes".cmTransferPnPLeftClampOpenClose.monitoring.inWorkPos;
   #statTonTime[130].TON(IN := #_w1 AND "Unit1.Em5.ControlNodes".transferPnPLeft."step".transition1[130],
                         PT := #delayTime);
   IF #statTonTime[130].Q THEN
       "Unit1.Em5.ControlNodes".transferPnPLeft.sequence.status.nextStep := #JOB_1_STEP_60;
   END_IF;
END_REGION

REGION Network 11: Step[160] : Transfer PP Left Y-Axis Wait Pos
   RUNG wire#powerrail
      { S7_Templates := "SrcType := DInt" } EQ_Contact(in1 := "Unit1.Em5.ControlNodes".transferPnPLeft.sequence.status.currentStep, in2 := #JOB_1_STEP_60)
      Contact( "Unit1.Em5.ControlNodes".transferPnPLeft.sequence.status.seqActive )
      wire#w1
      I_Contact( "Unit1.Em5.ControlNodes".cm.softcam.transferPnPLeftAxisY.pos00_wait.inPos )
      Coil( "Unit1.Em5.ControlNodes".transferPnPLeft."step".action1[160] )
   END_RUNG
   RUNG wire#w1
      Contact( "Unit1.Em5.ControlNodes".cm.softcam.transferPnPLeftAxisY.pos00_wait.inPos )
      Coil( "Unit1.Em5.ControlNodes".transferPnPLeft."step".transition1[160] )
   END_RUNG
   RUNG wire#w1
      Contact( "Unit1.Em5.ControlNodes".transferPnPLeft."step".transition1[160] )
      { S7_Templates := "time_type := Time" } #statTonTime[160].TON(pt := #delayTime, et =>)
      Move(in := #JOB_1_STEP_70, out1 => "Unit1.Em5.ControlNodes".transferPnPLeft.sequence.status.nextStep)
   END_RUNG
   // the same network as SCL:
   #_w1 := ("Unit1.Em5.ControlNodes".transferPnPLeft.sequence.status.currentStep = #JOB_1_STEP_60) AND "Unit1.Em5.ControlNodes".transferPnPLeft.sequence.status.seqActive;
   "Unit1.Em5.ControlNodes".transferPnPLeft."step".action1[160] := #_w1 AND NOT "Unit1.Em5.ControlNodes".cm.softcam.transferPnPLeftAxisY.pos00_wait.inPos;
   "Unit1.Em5.ControlNodes".transferPnPLeft."step".transition1[160] := #_w1 AND "Unit1.Em5.ControlNodes".cm.softcam.transferPnPLeftAxisY.pos00_wait.inPos;
   #statTonTime[160].TON(IN := #_w1 AND "Unit1.Em5.ControlNodes".transferPnPLeft."step".transition1[160],
                         PT := #delayTime);
   IF #statTonTime[160].Q THEN
       "Unit1.Em5.ControlNodes".transferPnPLeft.sequence.status.nextStep := #JOB_1_STEP_70;
   END_IF;
END_REGION

REGION Network 12: Step[170] : Transfer PP Left Z-Axis Wait Pos
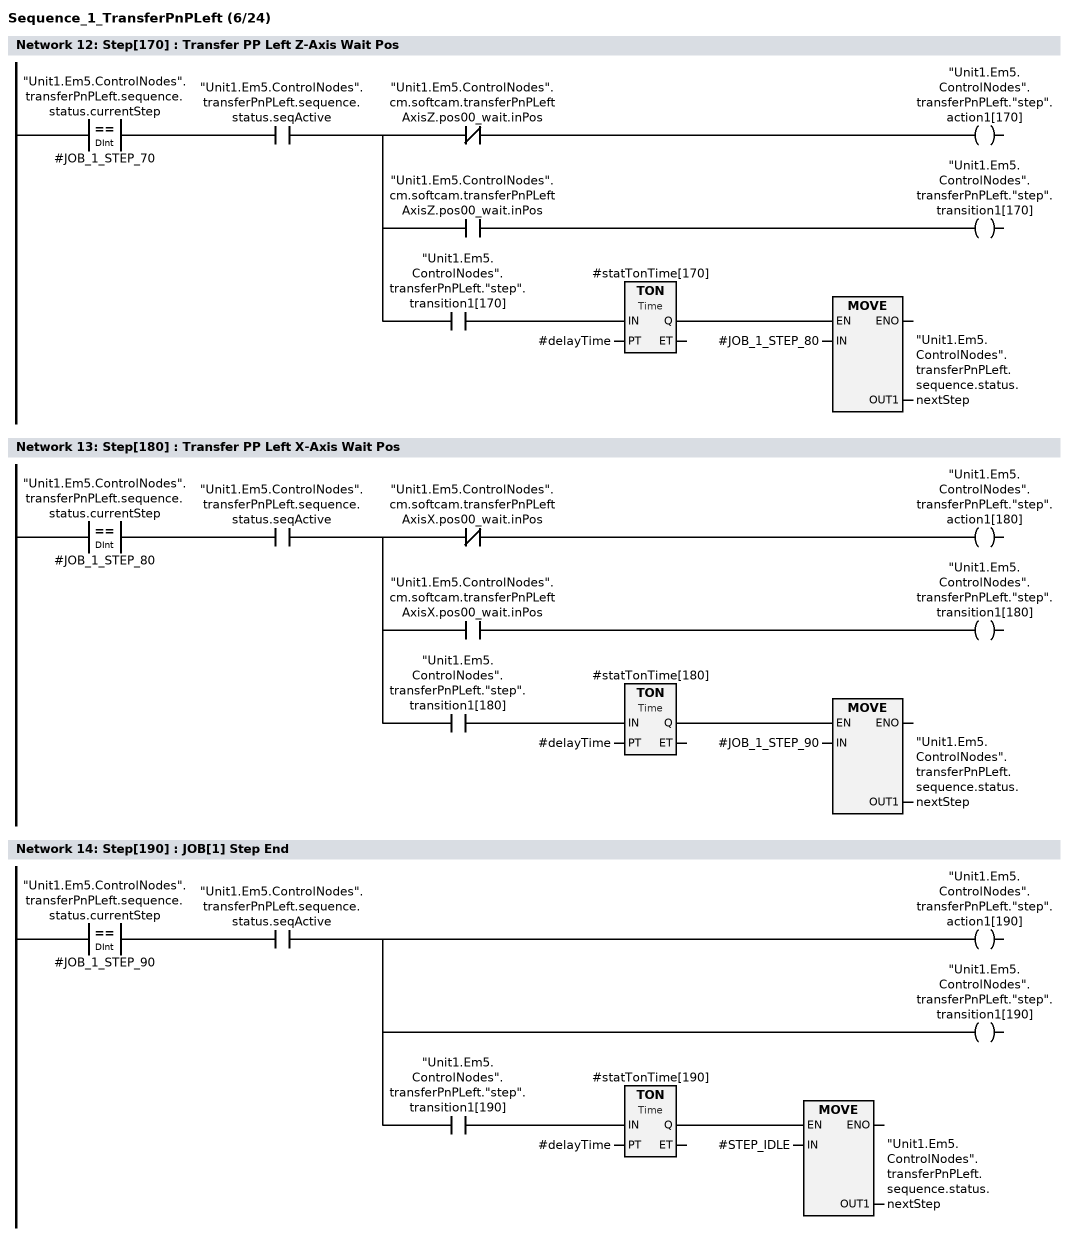
   RUNG wire#powerrail
      { S7_Templates := "SrcType := DInt" } EQ_Contact(in1 := "Unit1.Em5.ControlNodes".transferPnPLeft.sequence.status.currentStep, in2 := #JOB_1_STEP_70)
      Contact( "Unit1.Em5.ControlNodes".transferPnPLeft.sequence.status.seqActive )
      wire#w1
      I_Contact( "Unit1.Em5.ControlNodes".cm.softcam.transferPnPLeftAxisZ.pos00_wait.inPos )
      Coil( "Unit1.Em5.ControlNodes".transferPnPLeft."step".action1[170] )
   END_RUNG
   RUNG wire#w1
      Contact( "Unit1.Em5.ControlNodes".cm.softcam.transferPnPLeftAxisZ.pos00_wait.inPos )
      Coil( "Unit1.Em5.ControlNodes".transferPnPLeft."step".transition1[170] )
   END_RUNG
   RUNG wire#w1
      Contact( "Unit1.Em5.ControlNodes".transferPnPLeft."step".transition1[170] )
      { S7_Templates := "time_type := Time" } #statTonTime[170].TON(pt := #delayTime, et =>)
      Move(in := #JOB_1_STEP_80, out1 => "Unit1.Em5.ControlNodes".transferPnPLeft.sequence.status.nextStep)
   END_RUNG
   // the same network as SCL:
   #_w1 := ("Unit1.Em5.ControlNodes".transferPnPLeft.sequence.status.currentStep = #JOB_1_STEP_70) AND "Unit1.Em5.ControlNodes".transferPnPLeft.sequence.status.seqActive;
   "Unit1.Em5.ControlNodes".transferPnPLeft."step".action1[170] := #_w1 AND NOT "Unit1.Em5.ControlNodes".cm.softcam.transferPnPLeftAxisZ.pos00_wait.inPos;
   "Unit1.Em5.ControlNodes".transferPnPLeft."step".transition1[170] := #_w1 AND "Unit1.Em5.ControlNodes".cm.softcam.transferPnPLeftAxisZ.pos00_wait.inPos;
   #statTonTime[170].TON(IN := #_w1 AND "Unit1.Em5.ControlNodes".transferPnPLeft."step".transition1[170],
                         PT := #delayTime);
   IF #statTonTime[170].Q THEN
       "Unit1.Em5.ControlNodes".transferPnPLeft.sequence.status.nextStep := #JOB_1_STEP_80;
   END_IF;
END_REGION

REGION Network 13: Step[180] : Transfer PP Left X-Axis Wait Pos
   RUNG wire#powerrail
      { S7_Templates := "SrcType := DInt" } EQ_Contact(in1 := "Unit1.Em5.ControlNodes".transferPnPLeft.sequence.status.currentStep, in2 := #JOB_1_STEP_80)
      Contact( "Unit1.Em5.ControlNodes".transferPnPLeft.sequence.status.seqActive )
      wire#w1
      I_Contact( "Unit1.Em5.ControlNodes".cm.softcam.transferPnPLeftAxisX.pos00_wait.inPos )
      Coil( "Unit1.Em5.ControlNodes".transferPnPLeft."step".action1[180] )
   END_RUNG
   RUNG wire#w1
      Contact( "Unit1.Em5.ControlNodes".cm.softcam.transferPnPLeftAxisX.pos00_wait.inPos )
      Coil( "Unit1.Em5.ControlNodes".transferPnPLeft."step".transition1[180] )
   END_RUNG
   RUNG wire#w1
      Contact( "Unit1.Em5.ControlNodes".transferPnPLeft."step".transition1[180] )
      { S7_Templates := "time_type := Time" } #statTonTime[180].TON(pt := #delayTime, et =>)
      Move(in := #JOB_1_STEP_90, out1 => "Unit1.Em5.ControlNodes".transferPnPLeft.sequence.status.nextStep)
   END_RUNG
   // the same network as SCL:
   #_w1 := ("Unit1.Em5.ControlNodes".transferPnPLeft.sequence.status.currentStep = #JOB_1_STEP_80) AND "Unit1.Em5.ControlNodes".transferPnPLeft.sequence.status.seqActive;
   "Unit1.Em5.ControlNodes".transferPnPLeft."step".action1[180] := #_w1 AND NOT "Unit1.Em5.ControlNodes".cm.softcam.transferPnPLeftAxisX.pos00_wait.inPos;
   "Unit1.Em5.ControlNodes".transferPnPLeft."step".transition1[180] := #_w1 AND "Unit1.Em5.ControlNodes".cm.softcam.transferPnPLeftAxisX.pos00_wait.inPos;
   #statTonTime[180].TON(IN := #_w1 AND "Unit1.Em5.ControlNodes".transferPnPLeft."step".transition1[180],
                         PT := #delayTime);
   IF #statTonTime[180].Q THEN
       "Unit1.Em5.ControlNodes".transferPnPLeft.sequence.status.nextStep := #JOB_1_STEP_90;
   END_IF;
END_REGION

REGION Network 14: Step[190] : JOB[1] Step End
   RUNG wire#powerrail
      { S7_Templates := "SrcType := DInt" } EQ_Contact(in1 := "Unit1.Em5.ControlNodes".transferPnPLeft.sequence.status.currentStep, in2 := #JOB_1_STEP_90)
      Contact( "Unit1.Em5.ControlNodes".transferPnPLeft.sequence.status.seqActive )
      wire#w1
      Coil( "Unit1.Em5.ControlNodes".transferPnPLeft."step".action1[190] )
   END_RUNG
   RUNG wire#w1
      Coil( "Unit1.Em5.ControlNodes".transferPnPLeft."step".transition1[190] )
   END_RUNG
   RUNG wire#w1
      Contact( "Unit1.Em5.ControlNodes".transferPnPLeft."step".transition1[190] )
      { S7_Templates := "time_type := Time" } #statTonTime[190].TON(pt := #delayTime, et =>)
      Move(in := #STEP_IDLE, out1 => "Unit1.Em5.ControlNodes".transferPnPLeft.sequence.status.nextStep)
   END_RUNG
   // the same network as SCL:
   "Unit1.Em5.ControlNodes".transferPnPLeft."step".action1[190] := ("Unit1.Em5.ControlNodes".transferPnPLeft.sequence.status.currentStep = #JOB_1_STEP_90) AND "Unit1.Em5.ControlNodes".transferPnPLeft.sequence.status.seqActive;
   "Unit1.Em5.ControlNodes".transferPnPLeft."step".transition1[190] := ("Unit1.Em5.ControlNodes".transferPnPLeft.sequence.status.currentStep = #JOB_1_STEP_90) AND "Unit1.Em5.ControlNodes".transferPnPLeft.sequence.status.seqActive;
   #statTonTime[190].TON(IN := ("Unit1.Em5.ControlNodes".transferPnPLeft.sequence.status.currentStep = #JOB_1_STEP_90) AND "Unit1.Em5.ControlNodes".transferPnPLeft.sequence.status.seqActive AND "Unit1.Em5.ControlNodes".transferPnPLeft."step".transition1[190],
                         PT := #delayTime);
   IF #statTonTime[190].Q THEN
       "Unit1.Em5.ControlNodes".transferPnPLeft.sequence.status.nextStep := #STEP_IDLE;
   END_IF;
END_REGION

REGION Network 15: ************** JOB[2] SIDE TAPE JR GET=AUTO-[A] ***************
END_REGION

REGION Network 16: Step[201] : JOB[2] Condition
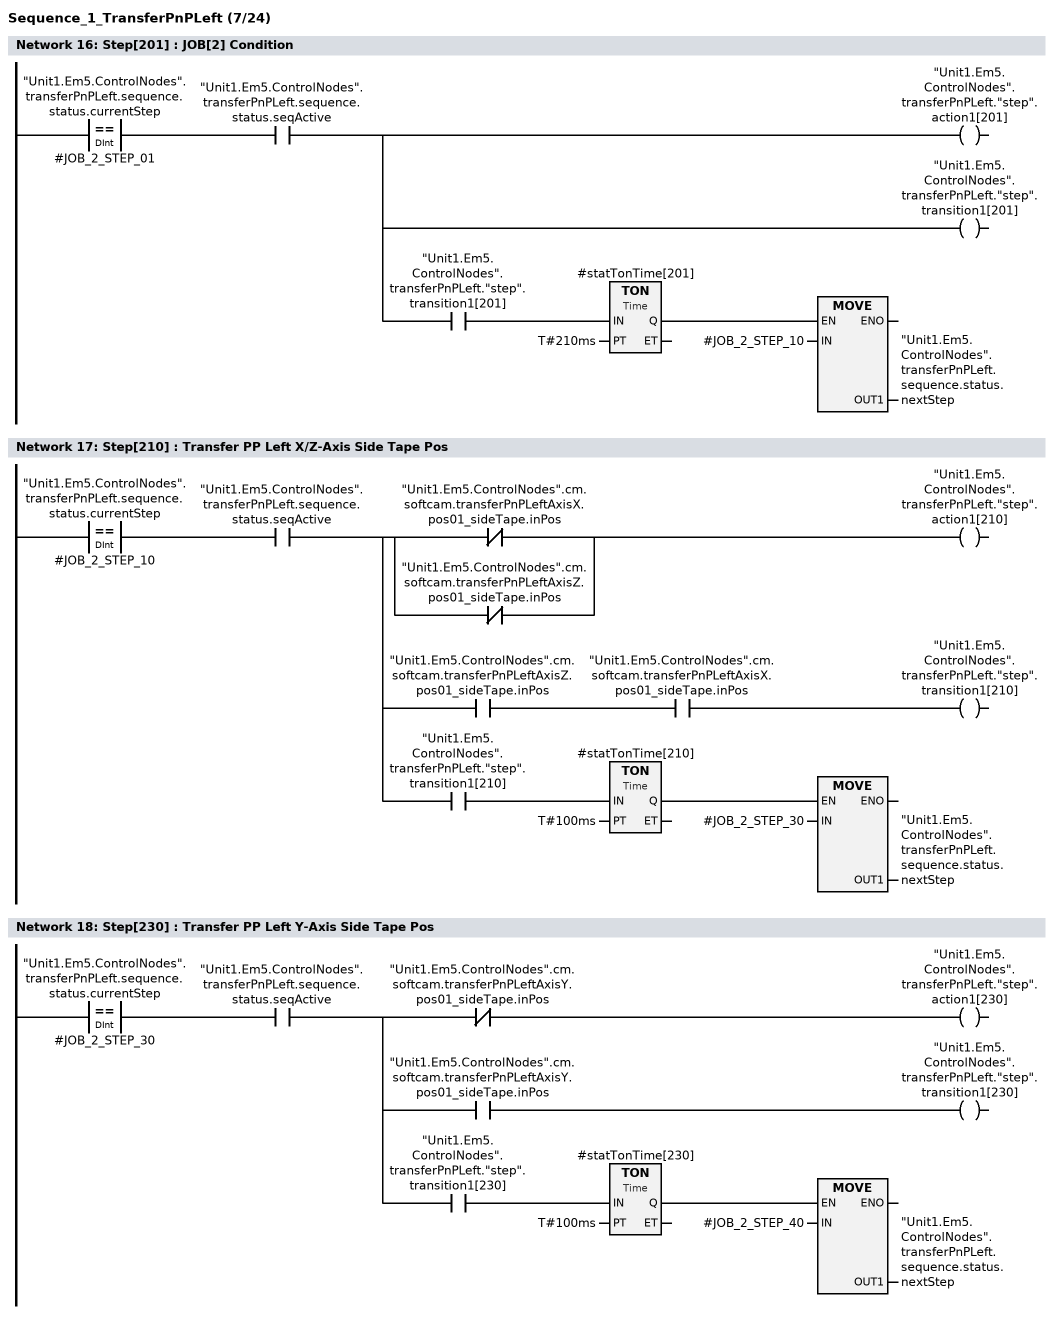
   RUNG wire#powerrail
      { S7_Templates := "SrcType := DInt" } EQ_Contact(in1 := "Unit1.Em5.ControlNodes".transferPnPLeft.sequence.status.currentStep, in2 := #JOB_2_STEP_01)
      Contact( "Unit1.Em5.ControlNodes".transferPnPLeft.sequence.status.seqActive )
      wire#w1
      Coil( "Unit1.Em5.ControlNodes".transferPnPLeft."step".action1[201] )
   END_RUNG
   RUNG wire#w1
      Coil( "Unit1.Em5.ControlNodes".transferPnPLeft."step".transition1[201] )
   END_RUNG
   RUNG wire#w1
      Contact( "Unit1.Em5.ControlNodes".transferPnPLeft."step".transition1[201] )
      { S7_Templates := "time_type := Time" } #statTonTime[201].TON(pt := T#210ms, et =>)
      Move(in := #JOB_2_STEP_10, out1 => "Unit1.Em5.ControlNodes".transferPnPLeft.sequence.status.nextStep)
   END_RUNG
   // the same network as SCL:
   "Unit1.Em5.ControlNodes".transferPnPLeft."step".action1[201] := ("Unit1.Em5.ControlNodes".transferPnPLeft.sequence.status.currentStep = #JOB_2_STEP_01) AND "Unit1.Em5.ControlNodes".transferPnPLeft.sequence.status.seqActive;
   "Unit1.Em5.ControlNodes".transferPnPLeft."step".transition1[201] := ("Unit1.Em5.ControlNodes".transferPnPLeft.sequence.status.currentStep = #JOB_2_STEP_01) AND "Unit1.Em5.ControlNodes".transferPnPLeft.sequence.status.seqActive;
   #statTonTime[201].TON(IN := ("Unit1.Em5.ControlNodes".transferPnPLeft.sequence.status.currentStep = #JOB_2_STEP_01) AND "Unit1.Em5.ControlNodes".transferPnPLeft.sequence.status.seqActive AND "Unit1.Em5.ControlNodes".transferPnPLeft."step".transition1[201],
                         PT := T#210ms);
   IF #statTonTime[201].Q THEN
       "Unit1.Em5.ControlNodes".transferPnPLeft.sequence.status.nextStep := #JOB_2_STEP_10;
   END_IF;
END_REGION

REGION Network 17: Step[210] : Transfer PP Left X/Z-Axis Side Tape Pos
   RUNG wire#powerrail
      { S7_Templates := "SrcType := DInt" } EQ_Contact(in1 := "Unit1.Em5.ControlNodes".transferPnPLeft.sequence.status.currentStep, in2 := #JOB_2_STEP_10)
      Contact( "Unit1.Em5.ControlNodes".transferPnPLeft.sequence.status.seqActive )
      wire#w1
      I_Contact( "Unit1.Em5.ControlNodes".cm.softcam.transferPnPLeftAxisX.pos01_sideTape.inPos )
      wire#w2
      Coil( "Unit1.Em5.ControlNodes".transferPnPLeft."step".action1[210] )
   END_RUNG
   RUNG wire#w1
      I_Contact( "Unit1.Em5.ControlNodes".cm.softcam.transferPnPLeftAxisZ.pos01_sideTape.inPos )
   END_RUNG wire#w2
   RUNG wire#w1
      Contact( "Unit1.Em5.ControlNodes".cm.softcam.transferPnPLeftAxisZ.pos01_sideTape.inPos )
      Contact( "Unit1.Em5.ControlNodes".cm.softcam.transferPnPLeftAxisX.pos01_sideTape.inPos )
      Coil( "Unit1.Em5.ControlNodes".transferPnPLeft."step".transition1[210] )
   END_RUNG
   RUNG wire#w1
      Contact( "Unit1.Em5.ControlNodes".transferPnPLeft."step".transition1[210] )
      { S7_Templates := "time_type := Time" } #statTonTime[210].TON(pt := T#100ms, et =>)
      Move(in := #JOB_2_STEP_30, out1 => "Unit1.Em5.ControlNodes".transferPnPLeft.sequence.status.nextStep)
   END_RUNG
   // the same network as SCL:
   #_w1 := ("Unit1.Em5.ControlNodes".transferPnPLeft.sequence.status.currentStep = #JOB_2_STEP_10) AND "Unit1.Em5.ControlNodes".transferPnPLeft.sequence.status.seqActive;
   "Unit1.Em5.ControlNodes".transferPnPLeft."step".action1[210] := #_w1 AND (NOT "Unit1.Em5.ControlNodes".cm.softcam.transferPnPLeftAxisX.pos01_sideTape.inPos OR NOT "Unit1.Em5.ControlNodes".cm.softcam.transferPnPLeftAxisZ.pos01_sideTape.inPos);
   "Unit1.Em5.ControlNodes".transferPnPLeft."step".transition1[210] := #_w1 AND "Unit1.Em5.ControlNodes".cm.softcam.transferPnPLeftAxisZ.pos01_sideTape.inPos AND "Unit1.Em5.ControlNodes".cm.softcam.transferPnPLeftAxisX.pos01_sideTape.inPos;
   #statTonTime[210].TON(IN := #_w1 AND "Unit1.Em5.ControlNodes".transferPnPLeft."step".transition1[210],
                         PT := T#100ms);
   IF #statTonTime[210].Q THEN
       "Unit1.Em5.ControlNodes".transferPnPLeft.sequence.status.nextStep := #JOB_2_STEP_30;
   END_IF;
END_REGION

REGION Network 18: Step[230] : Transfer PP Left Y-Axis Side Tape Pos
   RUNG wire#powerrail
      { S7_Templates := "SrcType := DInt" } EQ_Contact(in1 := "Unit1.Em5.ControlNodes".transferPnPLeft.sequence.status.currentStep, in2 := #JOB_2_STEP_30)
      Contact( "Unit1.Em5.ControlNodes".transferPnPLeft.sequence.status.seqActive )
      wire#w1
      I_Contact( "Unit1.Em5.ControlNodes".cm.softcam.transferPnPLeftAxisY.pos01_sideTape.inPos )
      Coil( "Unit1.Em5.ControlNodes".transferPnPLeft."step".action1[230] )
   END_RUNG
   RUNG wire#w1
      Contact( "Unit1.Em5.ControlNodes".cm.softcam.transferPnPLeftAxisY.pos01_sideTape.inPos )
      Coil( "Unit1.Em5.ControlNodes".transferPnPLeft."step".transition1[230] )
   END_RUNG
   RUNG wire#w1
      Contact( "Unit1.Em5.ControlNodes".transferPnPLeft."step".transition1[230] )
      { S7_Templates := "time_type := Time" } #statTonTime[230].TON(pt := T#100ms, et =>)
      Move(in := #JOB_2_STEP_40, out1 => "Unit1.Em5.ControlNodes".transferPnPLeft.sequence.status.nextStep)
   END_RUNG
   // the same network as SCL:
   #_w1 := ("Unit1.Em5.ControlNodes".transferPnPLeft.sequence.status.currentStep = #JOB_2_STEP_30) AND "Unit1.Em5.ControlNodes".transferPnPLeft.sequence.status.seqActive;
   "Unit1.Em5.ControlNodes".transferPnPLeft."step".action1[230] := #_w1 AND NOT "Unit1.Em5.ControlNodes".cm.softcam.transferPnPLeftAxisY.pos01_sideTape.inPos;
   "Unit1.Em5.ControlNodes".transferPnPLeft."step".transition1[230] := #_w1 AND "Unit1.Em5.ControlNodes".cm.softcam.transferPnPLeftAxisY.pos01_sideTape.inPos;
   #statTonTime[230].TON(IN := #_w1 AND "Unit1.Em5.ControlNodes".transferPnPLeft."step".transition1[230],
                         PT := T#100ms);
   IF #statTonTime[230].Q THEN
       "Unit1.Em5.ControlNodes".transferPnPLeft.sequence.status.nextStep := #JOB_2_STEP_40;
   END_IF;
END_REGION

REGION Network 19: Step[240] : Transfer PP Left Clamp Close
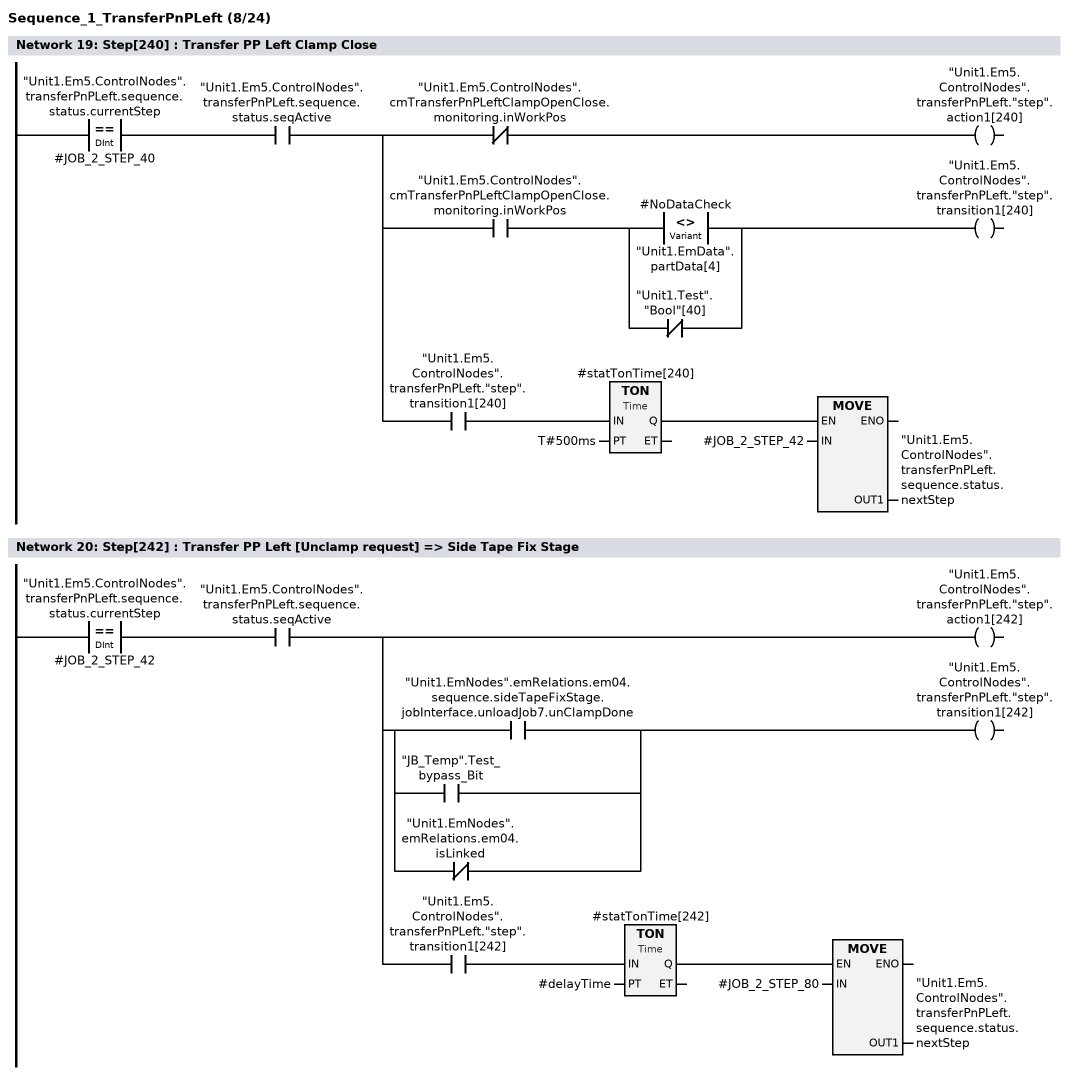
   RUNG wire#powerrail
      { S7_Templates := "SrcType := DInt" } EQ_Contact(in1 := "Unit1.Em5.ControlNodes".transferPnPLeft.sequence.status.currentStep, in2 := #JOB_2_STEP_40)
      Contact( "Unit1.Em5.ControlNodes".transferPnPLeft.sequence.status.seqActive )
      wire#w1
      I_Contact( "Unit1.Em5.ControlNodes".cmTransferPnPLeftClampOpenClose.monitoring.inWorkPos )
      Coil( "Unit1.Em5.ControlNodes".transferPnPLeft."step".action1[240] )
   END_RUNG
   RUNG wire#w1
      Contact( "Unit1.Em5.ControlNodes".cmTransferPnPLeftClampOpenClose.monitoring.inWorkPos )
      wire#w2
      { S7_Templates := "SrcType := Variant" } NE_Contact(in1 := #NoDataCheck, in2 := "Unit1.EmData".partData[4])
      wire#w3
      Coil( "Unit1.Em5.ControlNodes".transferPnPLeft."step".transition1[240] )
   END_RUNG
   RUNG wire#w2
      I_Contact( "Unit1.Test"."Bool"[40] )
   END_RUNG wire#w3
   RUNG wire#w1
      Contact( "Unit1.Em5.ControlNodes".transferPnPLeft."step".transition1[240] )
      { S7_Templates := "time_type := Time" } #statTonTime[240].TON(pt := T#500ms, et =>)
      Move(in := #JOB_2_STEP_42, out1 => "Unit1.Em5.ControlNodes".transferPnPLeft.sequence.status.nextStep)
   END_RUNG
   // the same network as SCL:
   #_w1 := ("Unit1.Em5.ControlNodes".transferPnPLeft.sequence.status.currentStep = #JOB_2_STEP_40) AND "Unit1.Em5.ControlNodes".transferPnPLeft.sequence.status.seqActive;
   "Unit1.Em5.ControlNodes".transferPnPLeft."step".action1[240] := #_w1 AND NOT "Unit1.Em5.ControlNodes".cmTransferPnPLeftClampOpenClose.monitoring.inWorkPos;
   "Unit1.Em5.ControlNodes".transferPnPLeft."step".transition1[240] := #_w1 AND "Unit1.Em5.ControlNodes".cmTransferPnPLeftClampOpenClose.monitoring.inWorkPos AND ((#NoDataCheck <> "Unit1.EmData".partData[4]) OR NOT "Unit1.Test"."Bool"[40]);
   #statTonTime[240].TON(IN := #_w1 AND "Unit1.Em5.ControlNodes".transferPnPLeft."step".transition1[240],
                         PT := T#500ms);
   IF #statTonTime[240].Q THEN
       "Unit1.Em5.ControlNodes".transferPnPLeft.sequence.status.nextStep := #JOB_2_STEP_42;
   END_IF;
END_REGION

REGION Network 20: Step[242] : Transfer PP Left [Unclamp request] => Side Tape Fix Stage
   RUNG wire#powerrail
      { S7_Templates := "SrcType := DInt" } EQ_Contact(in1 := "Unit1.Em5.ControlNodes".transferPnPLeft.sequence.status.currentStep, in2 := #JOB_2_STEP_42)
      Contact( "Unit1.Em5.ControlNodes".transferPnPLeft.sequence.status.seqActive )
      wire#w1
      Coil( "Unit1.Em5.ControlNodes".transferPnPLeft."step".action1[242] )
   END_RUNG
   RUNG wire#w1
      Contact( "Unit1.EmNodes".emRelations.em04.sequence.sideTapeFixStage.jobInterface.unloadJob7.unClampDone )
      wire#w2
      Coil( "Unit1.Em5.ControlNodes".transferPnPLeft."step".transition1[242] )
   END_RUNG
   RUNG wire#w1
      Contact( "JB_Temp".Test_bypass_Bit )
   END_RUNG wire#w2
   RUNG wire#w1
      I_Contact( "Unit1.EmNodes".emRelations.em04.isLinked )
   END_RUNG wire#w2
   RUNG wire#w1
      Contact( "Unit1.Em5.ControlNodes".transferPnPLeft."step".transition1[242] )
      { S7_Templates := "time_type := Time" } #statTonTime[242].TON(pt := #delayTime, et =>)
      Move(in := #JOB_2_STEP_80, out1 => "Unit1.Em5.ControlNodes".transferPnPLeft.sequence.status.nextStep)
   END_RUNG
   // the same network as SCL:
   "Unit1.Em5.ControlNodes".transferPnPLeft."step".action1[242] := ("Unit1.Em5.ControlNodes".transferPnPLeft.sequence.status.currentStep = #JOB_2_STEP_42) AND "Unit1.Em5.ControlNodes".transferPnPLeft.sequence.status.seqActive;
   "Unit1.Em5.ControlNodes".transferPnPLeft."step".transition1[242] := ("Unit1.Em5.ControlNodes".transferPnPLeft.sequence.status.currentStep = #JOB_2_STEP_42) AND "Unit1.Em5.ControlNodes".transferPnPLeft.sequence.status.seqActive AND ("Unit1.EmNodes".emRelations.em04.sequence.sideTapeFixStage.jobInterface.unloadJob7.unClampDone OR "JB_Temp".Test_bypass_Bit OR NOT "Unit1.EmNodes".emRelations.em04.isLinked);
   #statTonTime[242].TON(IN := ("Unit1.Em5.ControlNodes".transferPnPLeft.sequence.status.currentStep = #JOB_2_STEP_42) AND "Unit1.Em5.ControlNodes".transferPnPLeft.sequence.status.seqActive AND "Unit1.Em5.ControlNodes".transferPnPLeft."step".transition1[242],
                         PT := #delayTime);
   IF #statTonTime[242].Q THEN
       "Unit1.Em5.ControlNodes".transferPnPLeft.sequence.status.nextStep := #JOB_2_STEP_80;
   END_IF;
END_REGION

REGION Network 21: Step[280] : Transfer PP Left Y-Axis Wait Pos
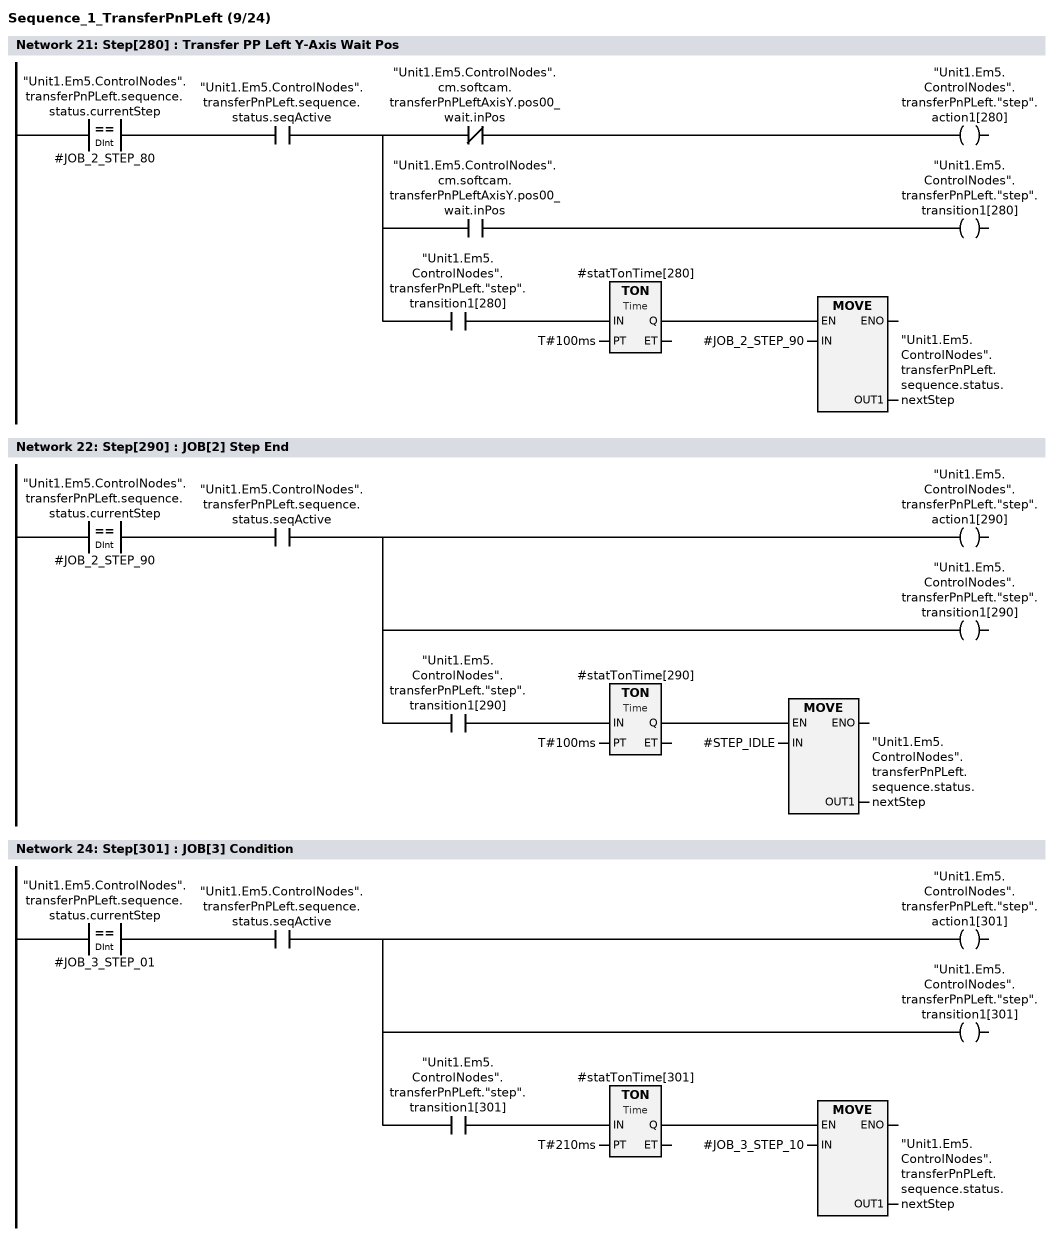
   RUNG wire#powerrail
      { S7_Templates := "SrcType := DInt" } EQ_Contact(in1 := "Unit1.Em5.ControlNodes".transferPnPLeft.sequence.status.currentStep, in2 := #JOB_2_STEP_80)
      Contact( "Unit1.Em5.ControlNodes".transferPnPLeft.sequence.status.seqActive )
      wire#w1
      I_Contact( "Unit1.Em5.ControlNodes".cm.softcam.transferPnPLeftAxisY.pos00_wait.inPos )
      Coil( "Unit1.Em5.ControlNodes".transferPnPLeft."step".action1[280] )
   END_RUNG
   RUNG wire#w1
      Contact( "Unit1.Em5.ControlNodes".cm.softcam.transferPnPLeftAxisY.pos00_wait.inPos )
      Coil( "Unit1.Em5.ControlNodes".transferPnPLeft."step".transition1[280] )
   END_RUNG
   RUNG wire#w1
      Contact( "Unit1.Em5.ControlNodes".transferPnPLeft."step".transition1[280] )
      { S7_Templates := "time_type := Time" } #statTonTime[280].TON(pt := T#100ms, et =>)
      Move(in := #JOB_2_STEP_90, out1 => "Unit1.Em5.ControlNodes".transferPnPLeft.sequence.status.nextStep)
   END_RUNG
   // the same network as SCL:
   #_w1 := ("Unit1.Em5.ControlNodes".transferPnPLeft.sequence.status.currentStep = #JOB_2_STEP_80) AND "Unit1.Em5.ControlNodes".transferPnPLeft.sequence.status.seqActive;
   "Unit1.Em5.ControlNodes".transferPnPLeft."step".action1[280] := #_w1 AND NOT "Unit1.Em5.ControlNodes".cm.softcam.transferPnPLeftAxisY.pos00_wait.inPos;
   "Unit1.Em5.ControlNodes".transferPnPLeft."step".transition1[280] := #_w1 AND "Unit1.Em5.ControlNodes".cm.softcam.transferPnPLeftAxisY.pos00_wait.inPos;
   #statTonTime[280].TON(IN := #_w1 AND "Unit1.Em5.ControlNodes".transferPnPLeft."step".transition1[280],
                         PT := T#100ms);
   IF #statTonTime[280].Q THEN
       "Unit1.Em5.ControlNodes".transferPnPLeft.sequence.status.nextStep := #JOB_2_STEP_90;
   END_IF;
END_REGION

REGION Network 22: Step[290] : JOB[2] Step End
   RUNG wire#powerrail
      { S7_Templates := "SrcType := DInt" } EQ_Contact(in1 := "Unit1.Em5.ControlNodes".transferPnPLeft.sequence.status.currentStep, in2 := #JOB_2_STEP_90)
      Contact( "Unit1.Em5.ControlNodes".transferPnPLeft.sequence.status.seqActive )
      wire#w1
      Coil( "Unit1.Em5.ControlNodes".transferPnPLeft."step".action1[290] )
   END_RUNG
   RUNG wire#w1
      Coil( "Unit1.Em5.ControlNodes".transferPnPLeft."step".transition1[290] )
   END_RUNG
   RUNG wire#w1
      Contact( "Unit1.Em5.ControlNodes".transferPnPLeft."step".transition1[290] )
      { S7_Templates := "time_type := Time" } #statTonTime[290].TON(pt := T#100ms, et =>)
      Move(in := #STEP_IDLE, out1 => "Unit1.Em5.ControlNodes".transferPnPLeft.sequence.status.nextStep)
   END_RUNG
   // the same network as SCL:
   "Unit1.Em5.ControlNodes".transferPnPLeft."step".action1[290] := ("Unit1.Em5.ControlNodes".transferPnPLeft.sequence.status.currentStep = #JOB_2_STEP_90) AND "Unit1.Em5.ControlNodes".transferPnPLeft.sequence.status.seqActive;
   "Unit1.Em5.ControlNodes".transferPnPLeft."step".transition1[290] := ("Unit1.Em5.ControlNodes".transferPnPLeft.sequence.status.currentStep = #JOB_2_STEP_90) AND "Unit1.Em5.ControlNodes".transferPnPLeft.sequence.status.seqActive;
   #statTonTime[290].TON(IN := ("Unit1.Em5.ControlNodes".transferPnPLeft.sequence.status.currentStep = #JOB_2_STEP_90) AND "Unit1.Em5.ControlNodes".transferPnPLeft.sequence.status.seqActive AND "Unit1.Em5.ControlNodes".transferPnPLeft."step".transition1[290],
                         PT := T#100ms);
   IF #statTonTime[290].Q THEN
       "Unit1.Em5.ControlNodes".transferPnPLeft.sequence.status.nextStep := #STEP_IDLE;
   END_IF;
END_REGION

REGION Network 23: ************ JOB[3] HOT PRESS LEFT JR PUT=AUTO-[A] *************
END_REGION

REGION Network 24: Step[301] : JOB[3] Condition
   RUNG wire#powerrail
      { S7_Templates := "SrcType := DInt" } EQ_Contact(in1 := "Unit1.Em5.ControlNodes".transferPnPLeft.sequence.status.currentStep, in2 := #JOB_3_STEP_01)
      Contact( "Unit1.Em5.ControlNodes".transferPnPLeft.sequence.status.seqActive )
      wire#w1
      Coil( "Unit1.Em5.ControlNodes".transferPnPLeft."step".action1[301] )
   END_RUNG
   RUNG wire#w1
      Coil( "Unit1.Em5.ControlNodes".transferPnPLeft."step".transition1[301] )
   END_RUNG
   RUNG wire#w1
      Contact( "Unit1.Em5.ControlNodes".transferPnPLeft."step".transition1[301] )
      { S7_Templates := "time_type := Time" } #statTonTime[301].TON(pt := T#210ms, et =>)
      Move(in := #JOB_3_STEP_10, out1 => "Unit1.Em5.ControlNodes".transferPnPLeft.sequence.status.nextStep)
   END_RUNG
   // the same network as SCL:
   "Unit1.Em5.ControlNodes".transferPnPLeft."step".action1[301] := ("Unit1.Em5.ControlNodes".transferPnPLeft.sequence.status.currentStep = #JOB_3_STEP_01) AND "Unit1.Em5.ControlNodes".transferPnPLeft.sequence.status.seqActive;
   "Unit1.Em5.ControlNodes".transferPnPLeft."step".transition1[301] := ("Unit1.Em5.ControlNodes".transferPnPLeft.sequence.status.currentStep = #JOB_3_STEP_01) AND "Unit1.Em5.ControlNodes".transferPnPLeft.sequence.status.seqActive;
   #statTonTime[301].TON(IN := ("Unit1.Em5.ControlNodes".transferPnPLeft.sequence.status.currentStep = #JOB_3_STEP_01) AND "Unit1.Em5.ControlNodes".transferPnPLeft.sequence.status.seqActive AND "Unit1.Em5.ControlNodes".transferPnPLeft."step".transition1[301],
                         PT := T#210ms);
   IF #statTonTime[301].Q THEN
       "Unit1.Em5.ControlNodes".transferPnPLeft.sequence.status.nextStep := #JOB_3_STEP_10;
   END_IF;
END_REGION

REGION Network 25: Step[310] : Transfer PP Left X/Z-Axis Hot Press Left Pos
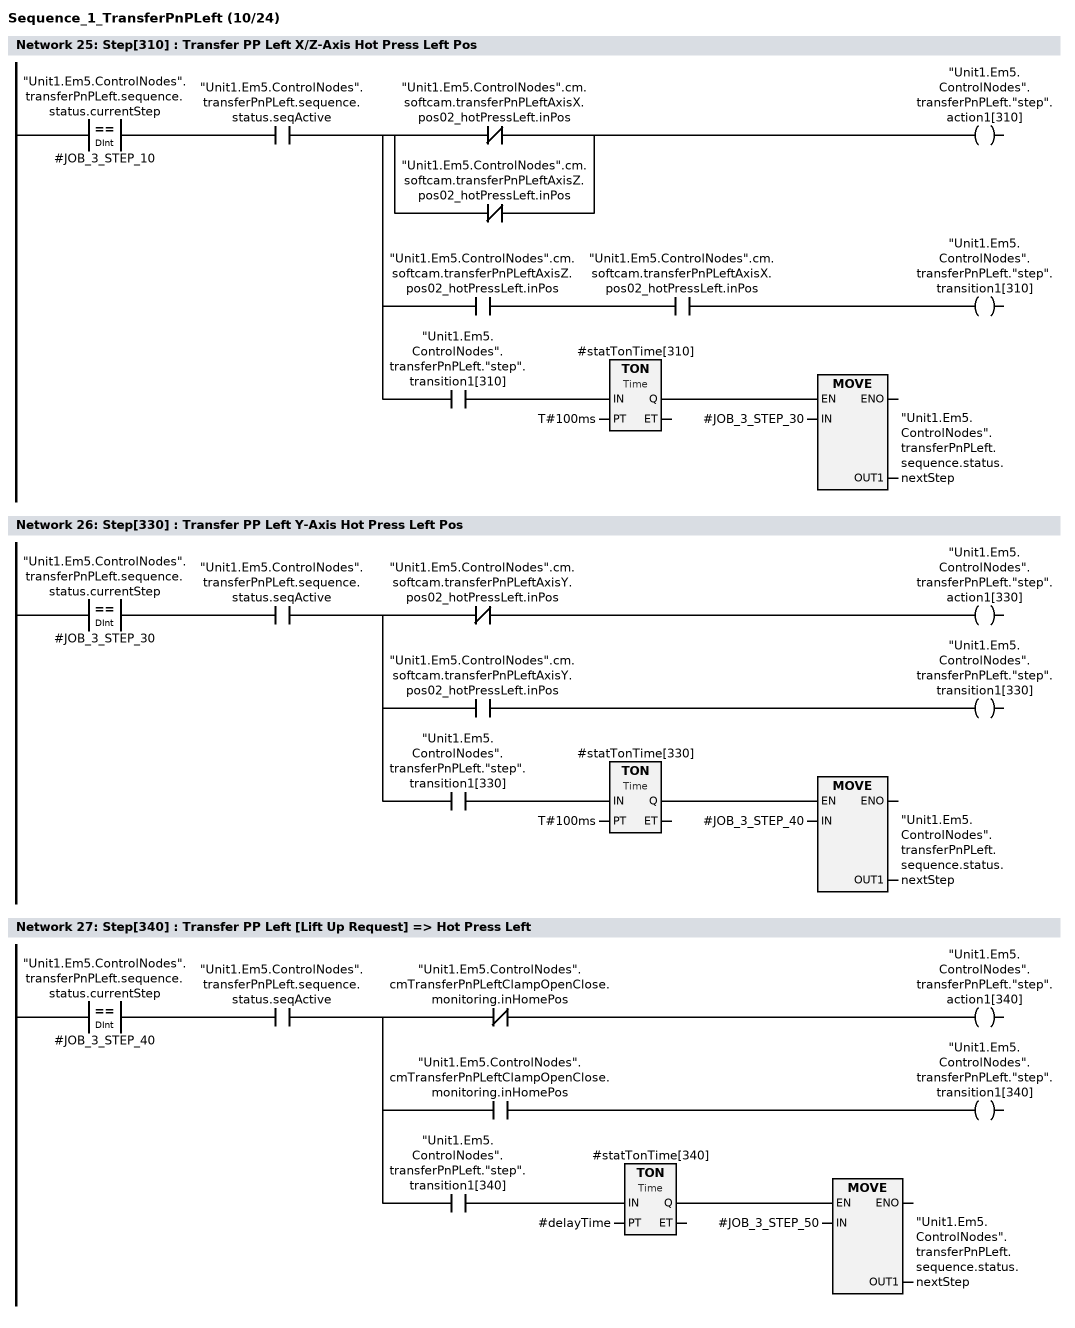
   RUNG wire#powerrail
      { S7_Templates := "SrcType := DInt" } EQ_Contact(in1 := "Unit1.Em5.ControlNodes".transferPnPLeft.sequence.status.currentStep, in2 := #JOB_3_STEP_10)
      Contact( "Unit1.Em5.ControlNodes".transferPnPLeft.sequence.status.seqActive )
      wire#w1
      I_Contact( "Unit1.Em5.ControlNodes".cm.softcam.transferPnPLeftAxisX.pos02_hotPressLeft.inPos )
      wire#w2
      Coil( "Unit1.Em5.ControlNodes".transferPnPLeft."step".action1[310] )
   END_RUNG
   RUNG wire#w1
      I_Contact( "Unit1.Em5.ControlNodes".cm.softcam.transferPnPLeftAxisZ.pos02_hotPressLeft.inPos )
   END_RUNG wire#w2
   RUNG wire#w1
      Contact( "Unit1.Em5.ControlNodes".cm.softcam.transferPnPLeftAxisZ.pos02_hotPressLeft.inPos )
      Contact( "Unit1.Em5.ControlNodes".cm.softcam.transferPnPLeftAxisX.pos02_hotPressLeft.inPos )
      Coil( "Unit1.Em5.ControlNodes".transferPnPLeft."step".transition1[310] )
   END_RUNG
   RUNG wire#w1
      Contact( "Unit1.Em5.ControlNodes".transferPnPLeft."step".transition1[310] )
      { S7_Templates := "time_type := Time" } #statTonTime[310].TON(pt := T#100ms, et =>)
      Move(in := #JOB_3_STEP_30, out1 => "Unit1.Em5.ControlNodes".transferPnPLeft.sequence.status.nextStep)
   END_RUNG
   // the same network as SCL:
   #_w1 := ("Unit1.Em5.ControlNodes".transferPnPLeft.sequence.status.currentStep = #JOB_3_STEP_10) AND "Unit1.Em5.ControlNodes".transferPnPLeft.sequence.status.seqActive;
   "Unit1.Em5.ControlNodes".transferPnPLeft."step".action1[310] := #_w1 AND (NOT "Unit1.Em5.ControlNodes".cm.softcam.transferPnPLeftAxisX.pos02_hotPressLeft.inPos OR NOT "Unit1.Em5.ControlNodes".cm.softcam.transferPnPLeftAxisZ.pos02_hotPressLeft.inPos);
   "Unit1.Em5.ControlNodes".transferPnPLeft."step".transition1[310] := #_w1 AND "Unit1.Em5.ControlNodes".cm.softcam.transferPnPLeftAxisZ.pos02_hotPressLeft.inPos AND "Unit1.Em5.ControlNodes".cm.softcam.transferPnPLeftAxisX.pos02_hotPressLeft.inPos;
   #statTonTime[310].TON(IN := #_w1 AND "Unit1.Em5.ControlNodes".transferPnPLeft."step".transition1[310],
                         PT := T#100ms);
   IF #statTonTime[310].Q THEN
       "Unit1.Em5.ControlNodes".transferPnPLeft.sequence.status.nextStep := #JOB_3_STEP_30;
   END_IF;
END_REGION

REGION Network 26: Step[330] : Transfer PP Left Y-Axis Hot Press Left Pos
   RUNG wire#powerrail
      { S7_Templates := "SrcType := DInt" } EQ_Contact(in1 := "Unit1.Em5.ControlNodes".transferPnPLeft.sequence.status.currentStep, in2 := #JOB_3_STEP_30)
      Contact( "Unit1.Em5.ControlNodes".transferPnPLeft.sequence.status.seqActive )
      wire#w1
      I_Contact( "Unit1.Em5.ControlNodes".cm.softcam.transferPnPLeftAxisY.pos02_hotPressLeft.inPos )
      Coil( "Unit1.Em5.ControlNodes".transferPnPLeft."step".action1[330] )
   END_RUNG
   RUNG wire#w1
      Contact( "Unit1.Em5.ControlNodes".cm.softcam.transferPnPLeftAxisY.pos02_hotPressLeft.inPos )
      Coil( "Unit1.Em5.ControlNodes".transferPnPLeft."step".transition1[330] )
   END_RUNG
   RUNG wire#w1
      Contact( "Unit1.Em5.ControlNodes".transferPnPLeft."step".transition1[330] )
      { S7_Templates := "time_type := Time" } #statTonTime[330].TON(pt := T#100ms, et =>)
      Move(in := #JOB_3_STEP_40, out1 => "Unit1.Em5.ControlNodes".transferPnPLeft.sequence.status.nextStep)
   END_RUNG
   // the same network as SCL:
   #_w1 := ("Unit1.Em5.ControlNodes".transferPnPLeft.sequence.status.currentStep = #JOB_3_STEP_30) AND "Unit1.Em5.ControlNodes".transferPnPLeft.sequence.status.seqActive;
   "Unit1.Em5.ControlNodes".transferPnPLeft."step".action1[330] := #_w1 AND NOT "Unit1.Em5.ControlNodes".cm.softcam.transferPnPLeftAxisY.pos02_hotPressLeft.inPos;
   "Unit1.Em5.ControlNodes".transferPnPLeft."step".transition1[330] := #_w1 AND "Unit1.Em5.ControlNodes".cm.softcam.transferPnPLeftAxisY.pos02_hotPressLeft.inPos;
   #statTonTime[330].TON(IN := #_w1 AND "Unit1.Em5.ControlNodes".transferPnPLeft."step".transition1[330],
                         PT := T#100ms);
   IF #statTonTime[330].Q THEN
       "Unit1.Em5.ControlNodes".transferPnPLeft.sequence.status.nextStep := #JOB_3_STEP_40;
   END_IF;
END_REGION

REGION Network 27: Step[340] : Transfer PP Left [Lift Up Request] => Hot Press Left
   RUNG wire#powerrail
      { S7_Templates := "SrcType := DInt" } EQ_Contact(in1 := "Unit1.Em5.ControlNodes".transferPnPLeft.sequence.status.currentStep, in2 := #JOB_3_STEP_40)
      Contact( "Unit1.Em5.ControlNodes".transferPnPLeft.sequence.status.seqActive )
      wire#w1
      I_Contact( "Unit1.Em5.ControlNodes".cmTransferPnPLeftClampOpenClose.monitoring.inHomePos )
      Coil( "Unit1.Em5.ControlNodes".transferPnPLeft."step".action1[340] )
   END_RUNG
   RUNG wire#w1
      Contact( "Unit1.Em5.ControlNodes".cmTransferPnPLeftClampOpenClose.monitoring.inHomePos )
      Coil( "Unit1.Em5.ControlNodes".transferPnPLeft."step".transition1[340] )
   END_RUNG
   RUNG wire#w1
      Contact( "Unit1.Em5.ControlNodes".transferPnPLeft."step".transition1[340] )
      { S7_Templates := "time_type := Time" } #statTonTime[340].TON(pt := #delayTime, et =>)
      Move(in := #JOB_3_STEP_50, out1 => "Unit1.Em5.ControlNodes".transferPnPLeft.sequence.status.nextStep)
   END_RUNG
   // the same network as SCL:
   #_w1 := ("Unit1.Em5.ControlNodes".transferPnPLeft.sequence.status.currentStep = #JOB_3_STEP_40) AND "Unit1.Em5.ControlNodes".transferPnPLeft.sequence.status.seqActive;
   "Unit1.Em5.ControlNodes".transferPnPLeft."step".action1[340] := #_w1 AND NOT "Unit1.Em5.ControlNodes".cmTransferPnPLeftClampOpenClose.monitoring.inHomePos;
   "Unit1.Em5.ControlNodes".transferPnPLeft."step".transition1[340] := #_w1 AND "Unit1.Em5.ControlNodes".cmTransferPnPLeftClampOpenClose.monitoring.inHomePos;
   #statTonTime[340].TON(IN := #_w1 AND "Unit1.Em5.ControlNodes".transferPnPLeft."step".transition1[340],
                         PT := #delayTime);
   IF #statTonTime[340].Q THEN
       "Unit1.Em5.ControlNodes".transferPnPLeft.sequence.status.nextStep := #JOB_3_STEP_50;
   END_IF;
END_REGION

REGION Network 28: Step[350] : Transfer PP Left Clamp Open
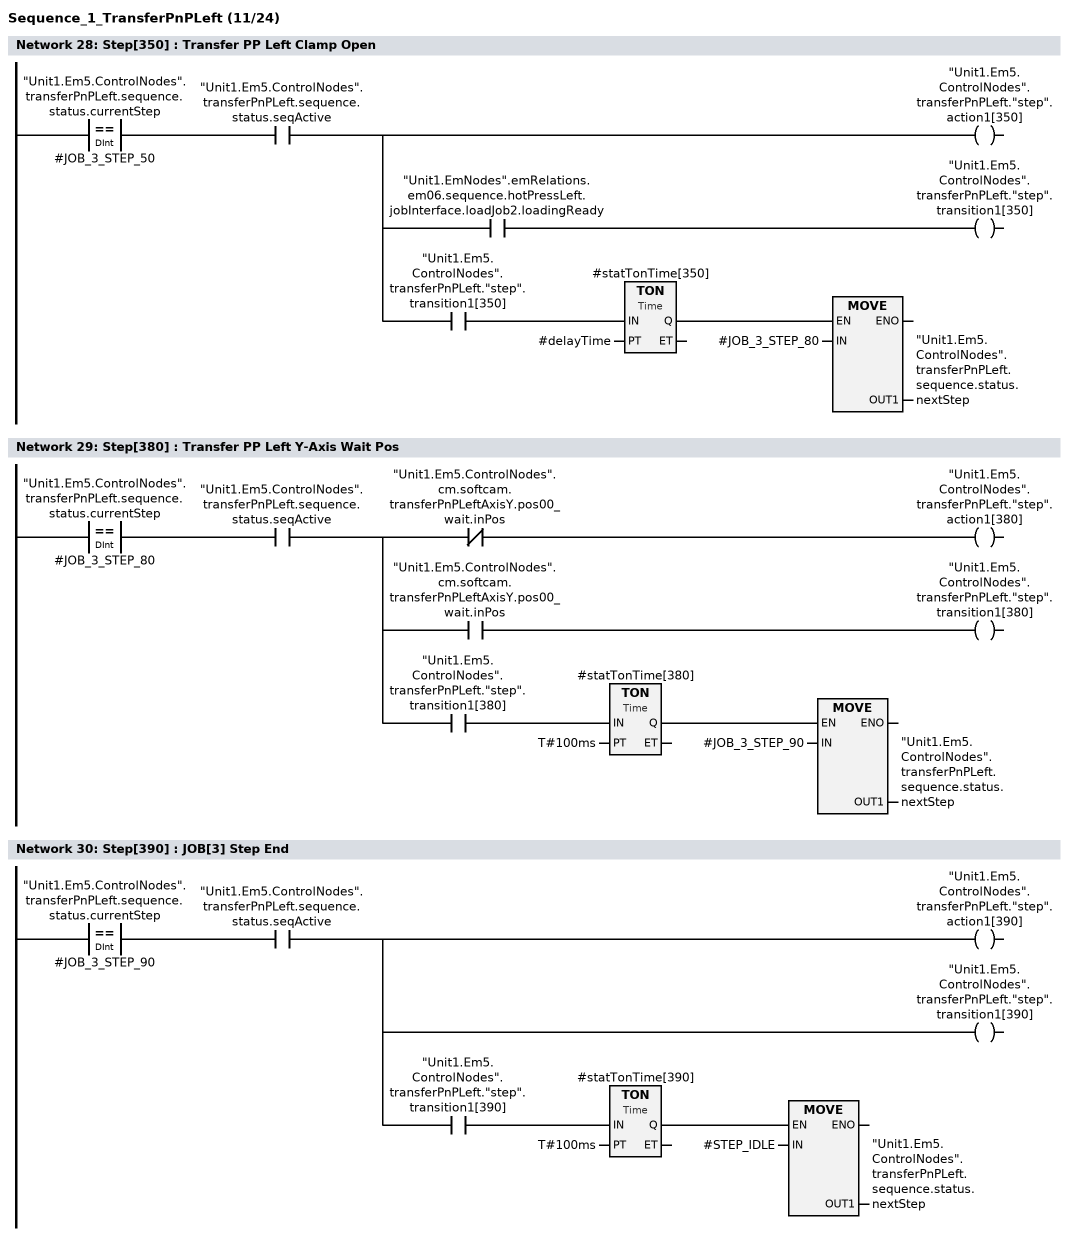
   RUNG wire#powerrail
      { S7_Templates := "SrcType := DInt" } EQ_Contact(in1 := "Unit1.Em5.ControlNodes".transferPnPLeft.sequence.status.currentStep, in2 := #JOB_3_STEP_50)
      Contact( "Unit1.Em5.ControlNodes".transferPnPLeft.sequence.status.seqActive )
      wire#w1
      Coil( "Unit1.Em5.ControlNodes".transferPnPLeft."step".action1[350] )
   END_RUNG
   RUNG wire#w1
      Contact( "Unit1.EmNodes".emRelations.em06.sequence.hotPressLeft.jobInterface.loadJob2.loadingReady )
      Coil( "Unit1.Em5.ControlNodes".transferPnPLeft."step".transition1[350] )
   END_RUNG
   RUNG wire#w1
      Contact( "Unit1.Em5.ControlNodes".transferPnPLeft."step".transition1[350] )
      { S7_Templates := "time_type := Time" } #statTonTime[350].TON(pt := #delayTime, et =>)
      Move(in := #JOB_3_STEP_80, out1 => "Unit1.Em5.ControlNodes".transferPnPLeft.sequence.status.nextStep)
   END_RUNG
   // the same network as SCL:
   "Unit1.Em5.ControlNodes".transferPnPLeft."step".action1[350] := ("Unit1.Em5.ControlNodes".transferPnPLeft.sequence.status.currentStep = #JOB_3_STEP_50) AND "Unit1.Em5.ControlNodes".transferPnPLeft.sequence.status.seqActive;
   "Unit1.Em5.ControlNodes".transferPnPLeft."step".transition1[350] := ("Unit1.Em5.ControlNodes".transferPnPLeft.sequence.status.currentStep = #JOB_3_STEP_50) AND "Unit1.Em5.ControlNodes".transferPnPLeft.sequence.status.seqActive AND "Unit1.EmNodes".emRelations.em06.sequence.hotPressLeft.jobInterface.loadJob2.loadingReady;
   #statTonTime[350].TON(IN := ("Unit1.Em5.ControlNodes".transferPnPLeft.sequence.status.currentStep = #JOB_3_STEP_50) AND "Unit1.Em5.ControlNodes".transferPnPLeft.sequence.status.seqActive AND "Unit1.Em5.ControlNodes".transferPnPLeft."step".transition1[350],
                         PT := #delayTime);
   IF #statTonTime[350].Q THEN
       "Unit1.Em5.ControlNodes".transferPnPLeft.sequence.status.nextStep := #JOB_3_STEP_80;
   END_IF;
END_REGION

REGION Network 29: Step[380] : Transfer PP Left Y-Axis Wait Pos
   RUNG wire#powerrail
      { S7_Templates := "SrcType := DInt" } EQ_Contact(in1 := "Unit1.Em5.ControlNodes".transferPnPLeft.sequence.status.currentStep, in2 := #JOB_3_STEP_80)
      Contact( "Unit1.Em5.ControlNodes".transferPnPLeft.sequence.status.seqActive )
      wire#w1
      I_Contact( "Unit1.Em5.ControlNodes".cm.softcam.transferPnPLeftAxisY.pos00_wait.inPos )
      Coil( "Unit1.Em5.ControlNodes".transferPnPLeft."step".action1[380] )
   END_RUNG
   RUNG wire#w1
      Contact( "Unit1.Em5.ControlNodes".cm.softcam.transferPnPLeftAxisY.pos00_wait.inPos )
      Coil( "Unit1.Em5.ControlNodes".transferPnPLeft."step".transition1[380] )
   END_RUNG
   RUNG wire#w1
      Contact( "Unit1.Em5.ControlNodes".transferPnPLeft."step".transition1[380] )
      { S7_Templates := "time_type := Time" } #statTonTime[380].TON(pt := T#100ms, et =>)
      Move(in := #JOB_3_STEP_90, out1 => "Unit1.Em5.ControlNodes".transferPnPLeft.sequence.status.nextStep)
   END_RUNG
   // the same network as SCL:
   #_w1 := ("Unit1.Em5.ControlNodes".transferPnPLeft.sequence.status.currentStep = #JOB_3_STEP_80) AND "Unit1.Em5.ControlNodes".transferPnPLeft.sequence.status.seqActive;
   "Unit1.Em5.ControlNodes".transferPnPLeft."step".action1[380] := #_w1 AND NOT "Unit1.Em5.ControlNodes".cm.softcam.transferPnPLeftAxisY.pos00_wait.inPos;
   "Unit1.Em5.ControlNodes".transferPnPLeft."step".transition1[380] := #_w1 AND "Unit1.Em5.ControlNodes".cm.softcam.transferPnPLeftAxisY.pos00_wait.inPos;
   #statTonTime[380].TON(IN := #_w1 AND "Unit1.Em5.ControlNodes".transferPnPLeft."step".transition1[380],
                         PT := T#100ms);
   IF #statTonTime[380].Q THEN
       "Unit1.Em5.ControlNodes".transferPnPLeft.sequence.status.nextStep := #JOB_3_STEP_90;
   END_IF;
END_REGION

REGION Network 30: Step[390] : JOB[3] Step End
   RUNG wire#powerrail
      { S7_Templates := "SrcType := DInt" } EQ_Contact(in1 := "Unit1.Em5.ControlNodes".transferPnPLeft.sequence.status.currentStep, in2 := #JOB_3_STEP_90)
      Contact( "Unit1.Em5.ControlNodes".transferPnPLeft.sequence.status.seqActive )
      wire#w1
      Coil( "Unit1.Em5.ControlNodes".transferPnPLeft."step".action1[390] )
   END_RUNG
   RUNG wire#w1
      Coil( "Unit1.Em5.ControlNodes".transferPnPLeft."step".transition1[390] )
   END_RUNG
   RUNG wire#w1
      Contact( "Unit1.Em5.ControlNodes".transferPnPLeft."step".transition1[390] )
      { S7_Templates := "time_type := Time" } #statTonTime[390].TON(pt := T#100ms, et =>)
      Move(in := #STEP_IDLE, out1 => "Unit1.Em5.ControlNodes".transferPnPLeft.sequence.status.nextStep)
   END_RUNG
   // the same network as SCL:
   "Unit1.Em5.ControlNodes".transferPnPLeft."step".action1[390] := ("Unit1.Em5.ControlNodes".transferPnPLeft.sequence.status.currentStep = #JOB_3_STEP_90) AND "Unit1.Em5.ControlNodes".transferPnPLeft.sequence.status.seqActive;
   "Unit1.Em5.ControlNodes".transferPnPLeft."step".transition1[390] := ("Unit1.Em5.ControlNodes".transferPnPLeft.sequence.status.currentStep = #JOB_3_STEP_90) AND "Unit1.Em5.ControlNodes".transferPnPLeft.sequence.status.seqActive;
   #statTonTime[390].TON(IN := ("Unit1.Em5.ControlNodes".transferPnPLeft.sequence.status.currentStep = #JOB_3_STEP_90) AND "Unit1.Em5.ControlNodes".transferPnPLeft.sequence.status.seqActive AND "Unit1.Em5.ControlNodes".transferPnPLeft."step".transition1[390],
                         PT := T#100ms);
   IF #statTonTime[390].Q THEN
       "Unit1.Em5.ControlNodes".transferPnPLeft.sequence.status.nextStep := #STEP_IDLE;
   END_IF;
END_REGION

REGION Network 31: ************ JOB[4] HOT PRESS LEFT JR GET=AUTO-[A] *************
END_REGION

REGION Network 32: Step[401] : JOB[4] Condition
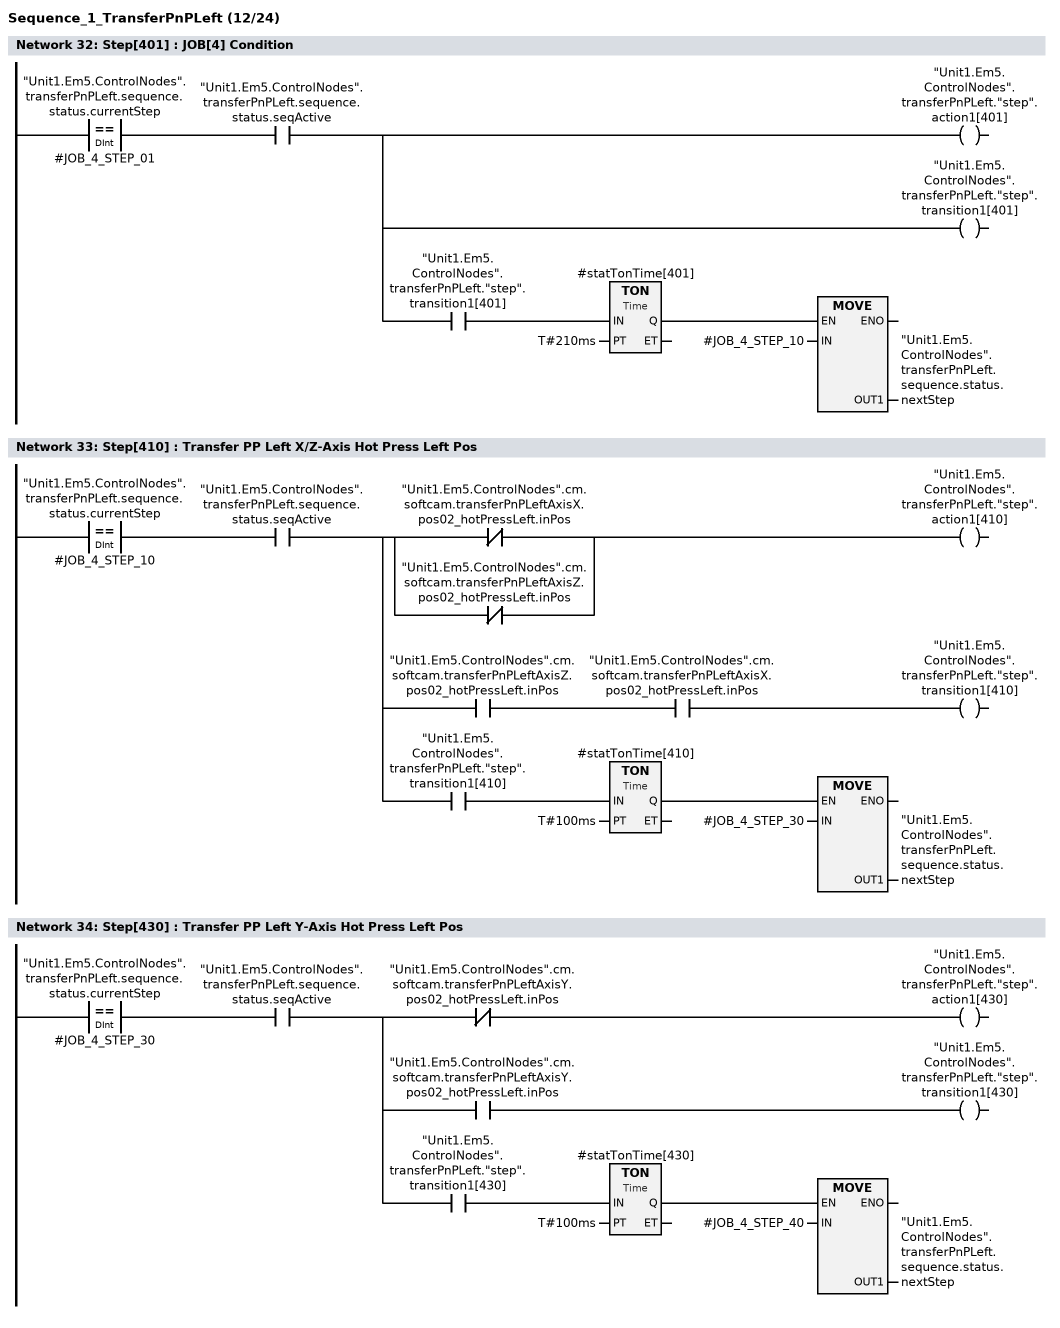
   RUNG wire#powerrail
      { S7_Templates := "SrcType := DInt" } EQ_Contact(in1 := "Unit1.Em5.ControlNodes".transferPnPLeft.sequence.status.currentStep, in2 := #JOB_4_STEP_01)
      Contact( "Unit1.Em5.ControlNodes".transferPnPLeft.sequence.status.seqActive )
      wire#w1
      Coil( "Unit1.Em5.ControlNodes".transferPnPLeft."step".action1[401] )
   END_RUNG
   RUNG wire#w1
      Coil( "Unit1.Em5.ControlNodes".transferPnPLeft."step".transition1[401] )
   END_RUNG
   RUNG wire#w1
      Contact( "Unit1.Em5.ControlNodes".transferPnPLeft."step".transition1[401] )
      { S7_Templates := "time_type := Time" } #statTonTime[401].TON(pt := T#210ms, et =>)
      Move(in := #JOB_4_STEP_10, out1 => "Unit1.Em5.ControlNodes".transferPnPLeft.sequence.status.nextStep)
   END_RUNG
   // the same network as SCL:
   "Unit1.Em5.ControlNodes".transferPnPLeft."step".action1[401] := ("Unit1.Em5.ControlNodes".transferPnPLeft.sequence.status.currentStep = #JOB_4_STEP_01) AND "Unit1.Em5.ControlNodes".transferPnPLeft.sequence.status.seqActive;
   "Unit1.Em5.ControlNodes".transferPnPLeft."step".transition1[401] := ("Unit1.Em5.ControlNodes".transferPnPLeft.sequence.status.currentStep = #JOB_4_STEP_01) AND "Unit1.Em5.ControlNodes".transferPnPLeft.sequence.status.seqActive;
   #statTonTime[401].TON(IN := ("Unit1.Em5.ControlNodes".transferPnPLeft.sequence.status.currentStep = #JOB_4_STEP_01) AND "Unit1.Em5.ControlNodes".transferPnPLeft.sequence.status.seqActive AND "Unit1.Em5.ControlNodes".transferPnPLeft."step".transition1[401],
                         PT := T#210ms);
   IF #statTonTime[401].Q THEN
       "Unit1.Em5.ControlNodes".transferPnPLeft.sequence.status.nextStep := #JOB_4_STEP_10;
   END_IF;
END_REGION

REGION Network 33: Step[410] : Transfer PP Left X/Z-Axis Hot Press Left Pos
   RUNG wire#powerrail
      { S7_Templates := "SrcType := DInt" } EQ_Contact(in1 := "Unit1.Em5.ControlNodes".transferPnPLeft.sequence.status.currentStep, in2 := #JOB_4_STEP_10)
      Contact( "Unit1.Em5.ControlNodes".transferPnPLeft.sequence.status.seqActive )
      wire#w1
      I_Contact( "Unit1.Em5.ControlNodes".cm.softcam.transferPnPLeftAxisX.pos02_hotPressLeft.inPos )
      wire#w2
      Coil( "Unit1.Em5.ControlNodes".transferPnPLeft."step".action1[410] )
   END_RUNG
   RUNG wire#w1
      I_Contact( "Unit1.Em5.ControlNodes".cm.softcam.transferPnPLeftAxisZ.pos02_hotPressLeft.inPos )
   END_RUNG wire#w2
   RUNG wire#w1
      Contact( "Unit1.Em5.ControlNodes".cm.softcam.transferPnPLeftAxisZ.pos02_hotPressLeft.inPos )
      Contact( "Unit1.Em5.ControlNodes".cm.softcam.transferPnPLeftAxisX.pos02_hotPressLeft.inPos )
      Coil( "Unit1.Em5.ControlNodes".transferPnPLeft."step".transition1[410] )
   END_RUNG
   RUNG wire#w1
      Contact( "Unit1.Em5.ControlNodes".transferPnPLeft."step".transition1[410] )
      { S7_Templates := "time_type := Time" } #statTonTime[410].TON(pt := T#100ms, et =>)
      Move(in := #JOB_4_STEP_30, out1 => "Unit1.Em5.ControlNodes".transferPnPLeft.sequence.status.nextStep)
   END_RUNG
   // the same network as SCL:
   #_w1 := ("Unit1.Em5.ControlNodes".transferPnPLeft.sequence.status.currentStep = #JOB_4_STEP_10) AND "Unit1.Em5.ControlNodes".transferPnPLeft.sequence.status.seqActive;
   "Unit1.Em5.ControlNodes".transferPnPLeft."step".action1[410] := #_w1 AND (NOT "Unit1.Em5.ControlNodes".cm.softcam.transferPnPLeftAxisX.pos02_hotPressLeft.inPos OR NOT "Unit1.Em5.ControlNodes".cm.softcam.transferPnPLeftAxisZ.pos02_hotPressLeft.inPos);
   "Unit1.Em5.ControlNodes".transferPnPLeft."step".transition1[410] := #_w1 AND "Unit1.Em5.ControlNodes".cm.softcam.transferPnPLeftAxisZ.pos02_hotPressLeft.inPos AND "Unit1.Em5.ControlNodes".cm.softcam.transferPnPLeftAxisX.pos02_hotPressLeft.inPos;
   #statTonTime[410].TON(IN := #_w1 AND "Unit1.Em5.ControlNodes".transferPnPLeft."step".transition1[410],
                         PT := T#100ms);
   IF #statTonTime[410].Q THEN
       "Unit1.Em5.ControlNodes".transferPnPLeft.sequence.status.nextStep := #JOB_4_STEP_30;
   END_IF;
END_REGION

REGION Network 34: Step[430] : Transfer PP Left Y-Axis Hot Press Left Pos
   RUNG wire#powerrail
      { S7_Templates := "SrcType := DInt" } EQ_Contact(in1 := "Unit1.Em5.ControlNodes".transferPnPLeft.sequence.status.currentStep, in2 := #JOB_4_STEP_30)
      Contact( "Unit1.Em5.ControlNodes".transferPnPLeft.sequence.status.seqActive )
      wire#w1
      I_Contact( "Unit1.Em5.ControlNodes".cm.softcam.transferPnPLeftAxisY.pos02_hotPressLeft.inPos )
      Coil( "Unit1.Em5.ControlNodes".transferPnPLeft."step".action1[430] )
   END_RUNG
   RUNG wire#w1
      Contact( "Unit1.Em5.ControlNodes".cm.softcam.transferPnPLeftAxisY.pos02_hotPressLeft.inPos )
      Coil( "Unit1.Em5.ControlNodes".transferPnPLeft."step".transition1[430] )
   END_RUNG
   RUNG wire#w1
      Contact( "Unit1.Em5.ControlNodes".transferPnPLeft."step".transition1[430] )
      { S7_Templates := "time_type := Time" } #statTonTime[430].TON(pt := T#100ms, et =>)
      Move(in := #JOB_4_STEP_40, out1 => "Unit1.Em5.ControlNodes".transferPnPLeft.sequence.status.nextStep)
   END_RUNG
   // the same network as SCL:
   #_w1 := ("Unit1.Em5.ControlNodes".transferPnPLeft.sequence.status.currentStep = #JOB_4_STEP_30) AND "Unit1.Em5.ControlNodes".transferPnPLeft.sequence.status.seqActive;
   "Unit1.Em5.ControlNodes".transferPnPLeft."step".action1[430] := #_w1 AND NOT "Unit1.Em5.ControlNodes".cm.softcam.transferPnPLeftAxisY.pos02_hotPressLeft.inPos;
   "Unit1.Em5.ControlNodes".transferPnPLeft."step".transition1[430] := #_w1 AND "Unit1.Em5.ControlNodes".cm.softcam.transferPnPLeftAxisY.pos02_hotPressLeft.inPos;
   #statTonTime[430].TON(IN := #_w1 AND "Unit1.Em5.ControlNodes".transferPnPLeft."step".transition1[430],
                         PT := T#100ms);
   IF #statTonTime[430].Q THEN
       "Unit1.Em5.ControlNodes".transferPnPLeft.sequence.status.nextStep := #JOB_4_STEP_40;
   END_IF;
END_REGION

REGION Network 35: Step[440] : Transfer PP Left Clamp Close
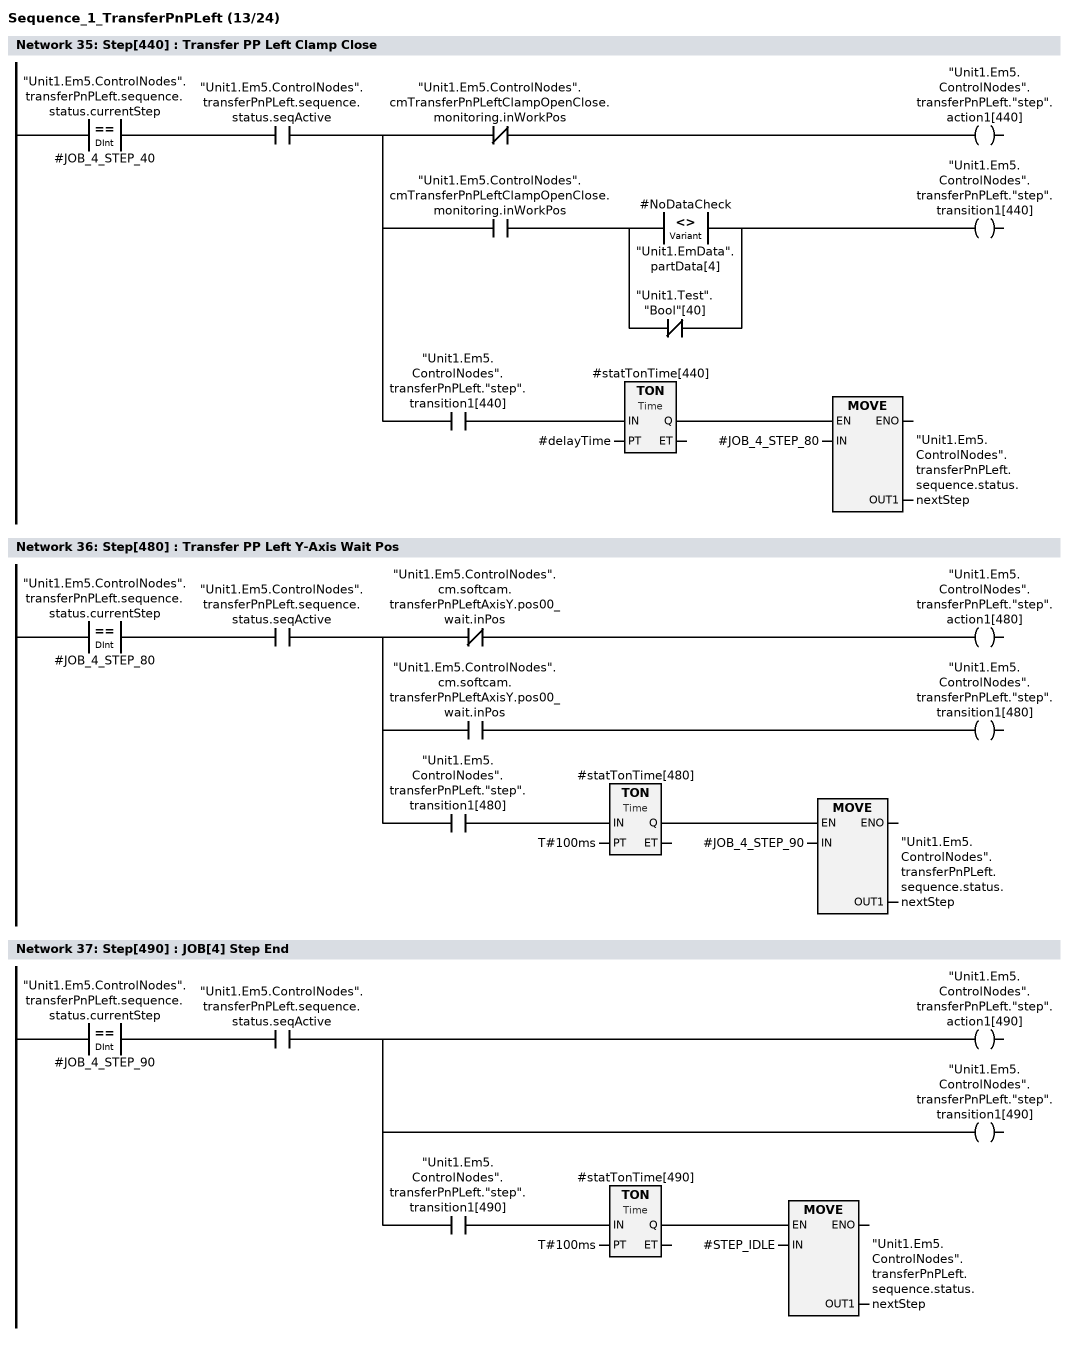
   RUNG wire#powerrail
      { S7_Templates := "SrcType := DInt" } EQ_Contact(in1 := "Unit1.Em5.ControlNodes".transferPnPLeft.sequence.status.currentStep, in2 := #JOB_4_STEP_40)
      Contact( "Unit1.Em5.ControlNodes".transferPnPLeft.sequence.status.seqActive )
      wire#w1
      I_Contact( "Unit1.Em5.ControlNodes".cmTransferPnPLeftClampOpenClose.monitoring.inWorkPos )
      Coil( "Unit1.Em5.ControlNodes".transferPnPLeft."step".action1[440] )
   END_RUNG
   RUNG wire#w1
      Contact( "Unit1.Em5.ControlNodes".cmTransferPnPLeftClampOpenClose.monitoring.inWorkPos )
      wire#w2
      { S7_Templates := "SrcType := Variant" } NE_Contact(in1 := #NoDataCheck, in2 := "Unit1.EmData".partData[4])
      wire#w3
      Coil( "Unit1.Em5.ControlNodes".transferPnPLeft."step".transition1[440] )
   END_RUNG
   RUNG wire#w2
      I_Contact( "Unit1.Test"."Bool"[40] )
   END_RUNG wire#w3
   RUNG wire#w1
      Contact( "Unit1.Em5.ControlNodes".transferPnPLeft."step".transition1[440] )
      { S7_Templates := "time_type := Time" } #statTonTime[440].TON(pt := #delayTime, et =>)
      Move(in := #JOB_4_STEP_80, out1 => "Unit1.Em5.ControlNodes".transferPnPLeft.sequence.status.nextStep)
   END_RUNG
   // the same network as SCL:
   #_w1 := ("Unit1.Em5.ControlNodes".transferPnPLeft.sequence.status.currentStep = #JOB_4_STEP_40) AND "Unit1.Em5.ControlNodes".transferPnPLeft.sequence.status.seqActive;
   "Unit1.Em5.ControlNodes".transferPnPLeft."step".action1[440] := #_w1 AND NOT "Unit1.Em5.ControlNodes".cmTransferPnPLeftClampOpenClose.monitoring.inWorkPos;
   "Unit1.Em5.ControlNodes".transferPnPLeft."step".transition1[440] := #_w1 AND "Unit1.Em5.ControlNodes".cmTransferPnPLeftClampOpenClose.monitoring.inWorkPos AND ((#NoDataCheck <> "Unit1.EmData".partData[4]) OR NOT "Unit1.Test"."Bool"[40]);
   #statTonTime[440].TON(IN := #_w1 AND "Unit1.Em5.ControlNodes".transferPnPLeft."step".transition1[440],
                         PT := #delayTime);
   IF #statTonTime[440].Q THEN
       "Unit1.Em5.ControlNodes".transferPnPLeft.sequence.status.nextStep := #JOB_4_STEP_80;
   END_IF;
END_REGION

REGION Network 36: Step[480] : Transfer PP Left Y-Axis Wait Pos
   RUNG wire#powerrail
      { S7_Templates := "SrcType := DInt" } EQ_Contact(in1 := "Unit1.Em5.ControlNodes".transferPnPLeft.sequence.status.currentStep, in2 := #JOB_4_STEP_80)
      Contact( "Unit1.Em5.ControlNodes".transferPnPLeft.sequence.status.seqActive )
      wire#w1
      I_Contact( "Unit1.Em5.ControlNodes".cm.softcam.transferPnPLeftAxisY.pos00_wait.inPos )
      Coil( "Unit1.Em5.ControlNodes".transferPnPLeft."step".action1[480] )
   END_RUNG
   RUNG wire#w1
      Contact( "Unit1.Em5.ControlNodes".cm.softcam.transferPnPLeftAxisY.pos00_wait.inPos )
      Coil( "Unit1.Em5.ControlNodes".transferPnPLeft."step".transition1[480] )
   END_RUNG
   RUNG wire#w1
      Contact( "Unit1.Em5.ControlNodes".transferPnPLeft."step".transition1[480] )
      { S7_Templates := "time_type := Time" } #statTonTime[480].TON(pt := T#100ms, et =>)
      Move(in := #JOB_4_STEP_90, out1 => "Unit1.Em5.ControlNodes".transferPnPLeft.sequence.status.nextStep)
   END_RUNG
   // the same network as SCL:
   #_w1 := ("Unit1.Em5.ControlNodes".transferPnPLeft.sequence.status.currentStep = #JOB_4_STEP_80) AND "Unit1.Em5.ControlNodes".transferPnPLeft.sequence.status.seqActive;
   "Unit1.Em5.ControlNodes".transferPnPLeft."step".action1[480] := #_w1 AND NOT "Unit1.Em5.ControlNodes".cm.softcam.transferPnPLeftAxisY.pos00_wait.inPos;
   "Unit1.Em5.ControlNodes".transferPnPLeft."step".transition1[480] := #_w1 AND "Unit1.Em5.ControlNodes".cm.softcam.transferPnPLeftAxisY.pos00_wait.inPos;
   #statTonTime[480].TON(IN := #_w1 AND "Unit1.Em5.ControlNodes".transferPnPLeft."step".transition1[480],
                         PT := T#100ms);
   IF #statTonTime[480].Q THEN
       "Unit1.Em5.ControlNodes".transferPnPLeft.sequence.status.nextStep := #JOB_4_STEP_90;
   END_IF;
END_REGION

REGION Network 37: Step[490] : JOB[4] Step End
   RUNG wire#powerrail
      { S7_Templates := "SrcType := DInt" } EQ_Contact(in1 := "Unit1.Em5.ControlNodes".transferPnPLeft.sequence.status.currentStep, in2 := #JOB_4_STEP_90)
      Contact( "Unit1.Em5.ControlNodes".transferPnPLeft.sequence.status.seqActive )
      wire#w1
      Coil( "Unit1.Em5.ControlNodes".transferPnPLeft."step".action1[490] )
   END_RUNG
   RUNG wire#w1
      Coil( "Unit1.Em5.ControlNodes".transferPnPLeft."step".transition1[490] )
   END_RUNG
   RUNG wire#w1
      Contact( "Unit1.Em5.ControlNodes".transferPnPLeft."step".transition1[490] )
      { S7_Templates := "time_type := Time" } #statTonTime[490].TON(pt := T#100ms, et =>)
      Move(in := #STEP_IDLE, out1 => "Unit1.Em5.ControlNodes".transferPnPLeft.sequence.status.nextStep)
   END_RUNG
   // the same network as SCL:
   "Unit1.Em5.ControlNodes".transferPnPLeft."step".action1[490] := ("Unit1.Em5.ControlNodes".transferPnPLeft.sequence.status.currentStep = #JOB_4_STEP_90) AND "Unit1.Em5.ControlNodes".transferPnPLeft.sequence.status.seqActive;
   "Unit1.Em5.ControlNodes".transferPnPLeft."step".transition1[490] := ("Unit1.Em5.ControlNodes".transferPnPLeft.sequence.status.currentStep = #JOB_4_STEP_90) AND "Unit1.Em5.ControlNodes".transferPnPLeft.sequence.status.seqActive;
   #statTonTime[490].TON(IN := ("Unit1.Em5.ControlNodes".transferPnPLeft.sequence.status.currentStep = #JOB_4_STEP_90) AND "Unit1.Em5.ControlNodes".transferPnPLeft.sequence.status.seqActive AND "Unit1.Em5.ControlNodes".transferPnPLeft."step".transition1[490],
                         PT := T#100ms);
   IF #statTonTime[490].Q THEN
       "Unit1.Em5.ControlNodes".transferPnPLeft.sequence.status.nextStep := #STEP_IDLE;
   END_IF;
END_REGION

REGION Network 38: ************** JOB[5] SIDE TAPE JR GET=AUTO-[B] ***************
END_REGION

REGION Network 39: Step[501] : JOB[5] Condition
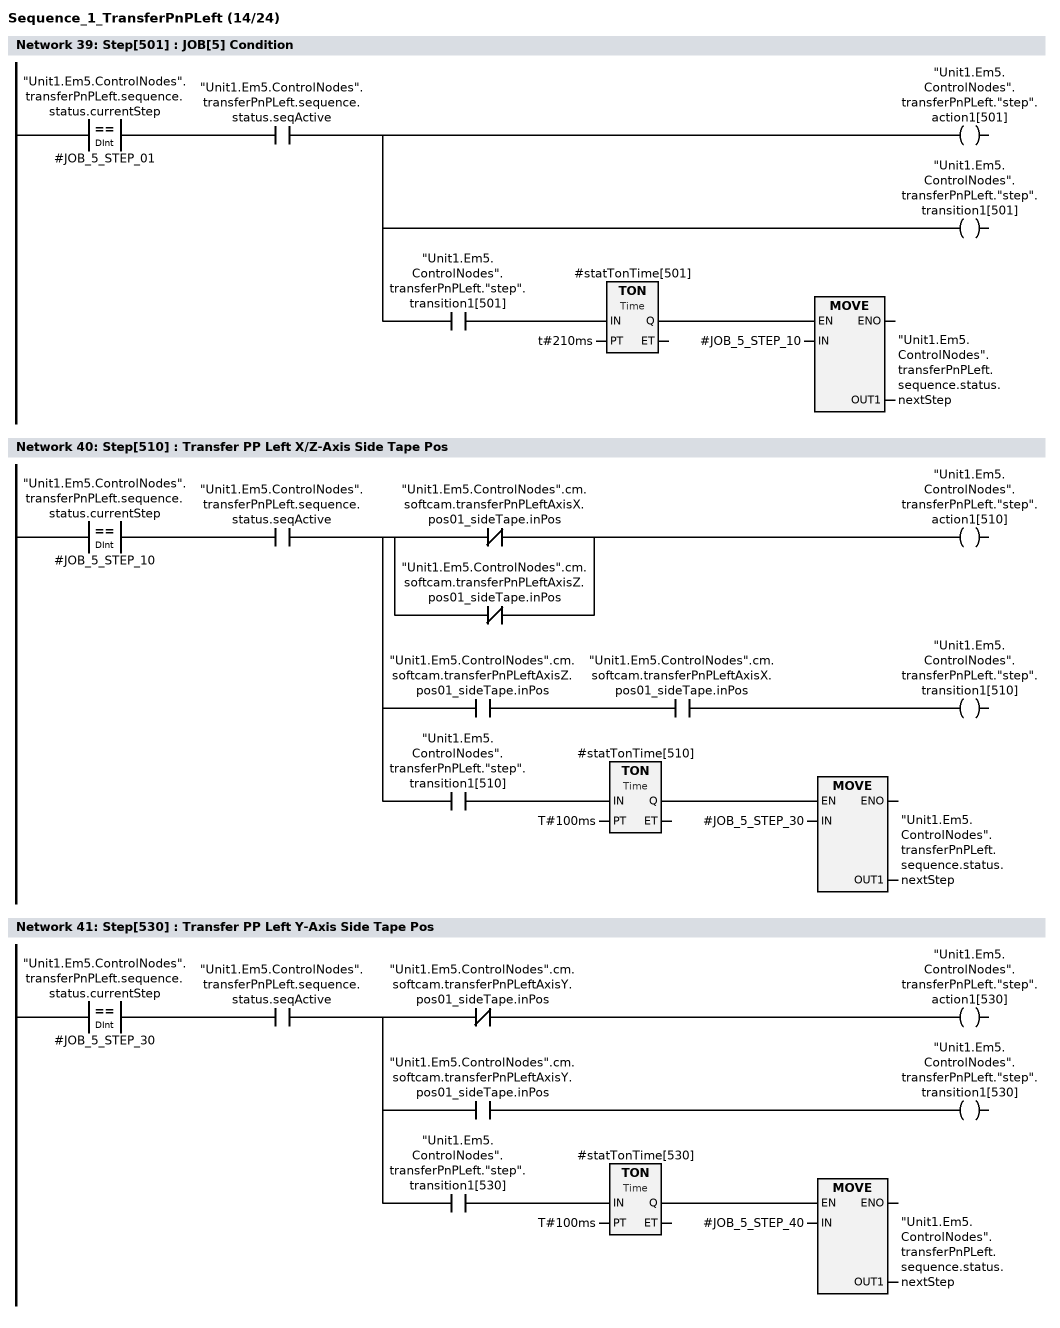
   RUNG wire#powerrail
      { S7_Templates := "SrcType := DInt" } EQ_Contact(in1 := "Unit1.Em5.ControlNodes".transferPnPLeft.sequence.status.currentStep, in2 := #JOB_5_STEP_01)
      Contact( "Unit1.Em5.ControlNodes".transferPnPLeft.sequence.status.seqActive )
      wire#w1
      Coil( "Unit1.Em5.ControlNodes".transferPnPLeft."step".action1[501] )
   END_RUNG
   RUNG wire#w1
      Coil( "Unit1.Em5.ControlNodes".transferPnPLeft."step".transition1[501] )
   END_RUNG
   RUNG wire#w1
      Contact( "Unit1.Em5.ControlNodes".transferPnPLeft."step".transition1[501] )
      { S7_Templates := "time_type := Time" } #statTonTime[501].TON(pt := t#210ms, et =>)
      Move(in := #JOB_5_STEP_10, out1 => "Unit1.Em5.ControlNodes".transferPnPLeft.sequence.status.nextStep)
   END_RUNG
   // the same network as SCL:
   "Unit1.Em5.ControlNodes".transferPnPLeft."step".action1[501] := ("Unit1.Em5.ControlNodes".transferPnPLeft.sequence.status.currentStep = #JOB_5_STEP_01) AND "Unit1.Em5.ControlNodes".transferPnPLeft.sequence.status.seqActive;
   "Unit1.Em5.ControlNodes".transferPnPLeft."step".transition1[501] := ("Unit1.Em5.ControlNodes".transferPnPLeft.sequence.status.currentStep = #JOB_5_STEP_01) AND "Unit1.Em5.ControlNodes".transferPnPLeft.sequence.status.seqActive;
   #statTonTime[501].TON(IN := ("Unit1.Em5.ControlNodes".transferPnPLeft.sequence.status.currentStep = #JOB_5_STEP_01) AND "Unit1.Em5.ControlNodes".transferPnPLeft.sequence.status.seqActive AND "Unit1.Em5.ControlNodes".transferPnPLeft."step".transition1[501],
                         PT := t#210ms);
   IF #statTonTime[501].Q THEN
       "Unit1.Em5.ControlNodes".transferPnPLeft.sequence.status.nextStep := #JOB_5_STEP_10;
   END_IF;
END_REGION

REGION Network 40: Step[510] : Transfer PP Left X/Z-Axis Side Tape Pos
   RUNG wire#powerrail
      { S7_Templates := "SrcType := DInt" } EQ_Contact(in1 := "Unit1.Em5.ControlNodes".transferPnPLeft.sequence.status.currentStep, in2 := #JOB_5_STEP_10)
      Contact( "Unit1.Em5.ControlNodes".transferPnPLeft.sequence.status.seqActive )
      wire#w1
      I_Contact( "Unit1.Em5.ControlNodes".cm.softcam.transferPnPLeftAxisX.pos01_sideTape.inPos )
      wire#w2
      Coil( "Unit1.Em5.ControlNodes".transferPnPLeft."step".action1[510] )
   END_RUNG
   RUNG wire#w1
      I_Contact( "Unit1.Em5.ControlNodes".cm.softcam.transferPnPLeftAxisZ.pos01_sideTape.inPos )
   END_RUNG wire#w2
   RUNG wire#w1
      Contact( "Unit1.Em5.ControlNodes".cm.softcam.transferPnPLeftAxisZ.pos01_sideTape.inPos )
      Contact( "Unit1.Em5.ControlNodes".cm.softcam.transferPnPLeftAxisX.pos01_sideTape.inPos )
      Coil( "Unit1.Em5.ControlNodes".transferPnPLeft."step".transition1[510] )
   END_RUNG
   RUNG wire#w1
      Contact( "Unit1.Em5.ControlNodes".transferPnPLeft."step".transition1[510] )
      { S7_Templates := "time_type := Time" } #statTonTime[510].TON(pt := T#100ms, et =>)
      Move(in := #JOB_5_STEP_30, out1 => "Unit1.Em5.ControlNodes".transferPnPLeft.sequence.status.nextStep)
   END_RUNG
   // the same network as SCL:
   #_w1 := ("Unit1.Em5.ControlNodes".transferPnPLeft.sequence.status.currentStep = #JOB_5_STEP_10) AND "Unit1.Em5.ControlNodes".transferPnPLeft.sequence.status.seqActive;
   "Unit1.Em5.ControlNodes".transferPnPLeft."step".action1[510] := #_w1 AND (NOT "Unit1.Em5.ControlNodes".cm.softcam.transferPnPLeftAxisX.pos01_sideTape.inPos OR NOT "Unit1.Em5.ControlNodes".cm.softcam.transferPnPLeftAxisZ.pos01_sideTape.inPos);
   "Unit1.Em5.ControlNodes".transferPnPLeft."step".transition1[510] := #_w1 AND "Unit1.Em5.ControlNodes".cm.softcam.transferPnPLeftAxisZ.pos01_sideTape.inPos AND "Unit1.Em5.ControlNodes".cm.softcam.transferPnPLeftAxisX.pos01_sideTape.inPos;
   #statTonTime[510].TON(IN := #_w1 AND "Unit1.Em5.ControlNodes".transferPnPLeft."step".transition1[510],
                         PT := T#100ms);
   IF #statTonTime[510].Q THEN
       "Unit1.Em5.ControlNodes".transferPnPLeft.sequence.status.nextStep := #JOB_5_STEP_30;
   END_IF;
END_REGION

REGION Network 41: Step[530] : Transfer PP Left Y-Axis Side Tape Pos
   RUNG wire#powerrail
      { S7_Templates := "SrcType := DInt" } EQ_Contact(in1 := "Unit1.Em5.ControlNodes".transferPnPLeft.sequence.status.currentStep, in2 := #JOB_5_STEP_30)
      Contact( "Unit1.Em5.ControlNodes".transferPnPLeft.sequence.status.seqActive )
      wire#w1
      I_Contact( "Unit1.Em5.ControlNodes".cm.softcam.transferPnPLeftAxisY.pos01_sideTape.inPos )
      Coil( "Unit1.Em5.ControlNodes".transferPnPLeft."step".action1[530] )
   END_RUNG
   RUNG wire#w1
      Contact( "Unit1.Em5.ControlNodes".cm.softcam.transferPnPLeftAxisY.pos01_sideTape.inPos )
      Coil( "Unit1.Em5.ControlNodes".transferPnPLeft."step".transition1[530] )
   END_RUNG
   RUNG wire#w1
      Contact( "Unit1.Em5.ControlNodes".transferPnPLeft."step".transition1[530] )
      { S7_Templates := "time_type := Time" } #statTonTime[530].TON(pt := T#100ms, et =>)
      Move(in := #JOB_5_STEP_40, out1 => "Unit1.Em5.ControlNodes".transferPnPLeft.sequence.status.nextStep)
   END_RUNG
   // the same network as SCL:
   #_w1 := ("Unit1.Em5.ControlNodes".transferPnPLeft.sequence.status.currentStep = #JOB_5_STEP_30) AND "Unit1.Em5.ControlNodes".transferPnPLeft.sequence.status.seqActive;
   "Unit1.Em5.ControlNodes".transferPnPLeft."step".action1[530] := #_w1 AND NOT "Unit1.Em5.ControlNodes".cm.softcam.transferPnPLeftAxisY.pos01_sideTape.inPos;
   "Unit1.Em5.ControlNodes".transferPnPLeft."step".transition1[530] := #_w1 AND "Unit1.Em5.ControlNodes".cm.softcam.transferPnPLeftAxisY.pos01_sideTape.inPos;
   #statTonTime[530].TON(IN := #_w1 AND "Unit1.Em5.ControlNodes".transferPnPLeft."step".transition1[530],
                         PT := T#100ms);
   IF #statTonTime[530].Q THEN
       "Unit1.Em5.ControlNodes".transferPnPLeft.sequence.status.nextStep := #JOB_5_STEP_40;
   END_IF;
END_REGION

REGION Network 42: Step[540] : Transfer PP Left Clamp Close
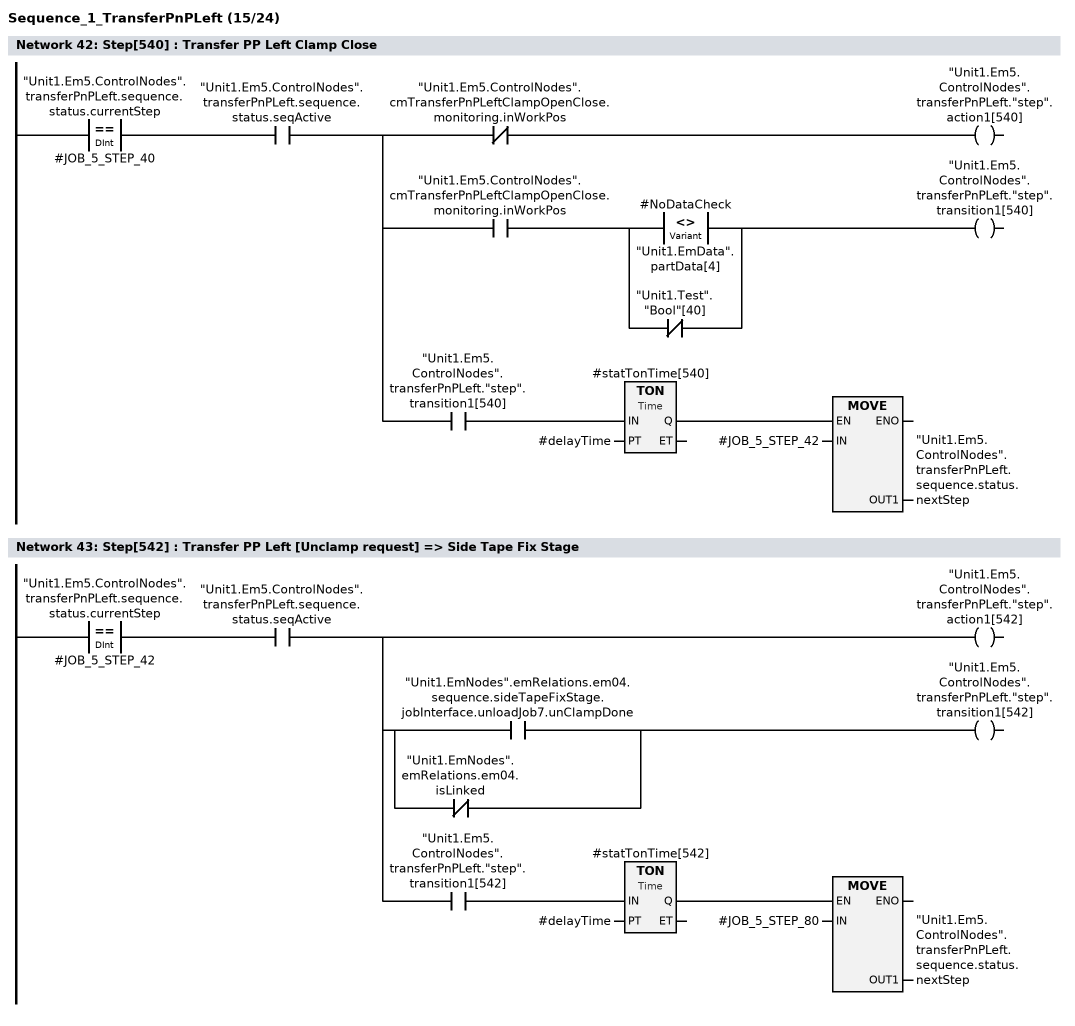
   RUNG wire#powerrail
      { S7_Templates := "SrcType := DInt" } EQ_Contact(in1 := "Unit1.Em5.ControlNodes".transferPnPLeft.sequence.status.currentStep, in2 := #JOB_5_STEP_40)
      Contact( "Unit1.Em5.ControlNodes".transferPnPLeft.sequence.status.seqActive )
      wire#w1
      I_Contact( "Unit1.Em5.ControlNodes".cmTransferPnPLeftClampOpenClose.monitoring.inWorkPos )
      Coil( "Unit1.Em5.ControlNodes".transferPnPLeft."step".action1[540] )
   END_RUNG
   RUNG wire#w1
      Contact( "Unit1.Em5.ControlNodes".cmTransferPnPLeftClampOpenClose.monitoring.inWorkPos )
      wire#w2
      { S7_Templates := "SrcType := Variant" } NE_Contact(in1 := #NoDataCheck, in2 := "Unit1.EmData".partData[4])
      wire#w3
      Coil( "Unit1.Em5.ControlNodes".transferPnPLeft."step".transition1[540] )
   END_RUNG
   RUNG wire#w2
      I_Contact( "Unit1.Test"."Bool"[40] )
   END_RUNG wire#w3
   RUNG wire#w1
      Contact( "Unit1.Em5.ControlNodes".transferPnPLeft."step".transition1[540] )
      { S7_Templates := "time_type := Time" } #statTonTime[540].TON(pt := #delayTime, et =>)
      Move(in := #JOB_5_STEP_42, out1 => "Unit1.Em5.ControlNodes".transferPnPLeft.sequence.status.nextStep)
   END_RUNG
   // the same network as SCL:
   #_w1 := ("Unit1.Em5.ControlNodes".transferPnPLeft.sequence.status.currentStep = #JOB_5_STEP_40) AND "Unit1.Em5.ControlNodes".transferPnPLeft.sequence.status.seqActive;
   "Unit1.Em5.ControlNodes".transferPnPLeft."step".action1[540] := #_w1 AND NOT "Unit1.Em5.ControlNodes".cmTransferPnPLeftClampOpenClose.monitoring.inWorkPos;
   "Unit1.Em5.ControlNodes".transferPnPLeft."step".transition1[540] := #_w1 AND "Unit1.Em5.ControlNodes".cmTransferPnPLeftClampOpenClose.monitoring.inWorkPos AND ((#NoDataCheck <> "Unit1.EmData".partData[4]) OR NOT "Unit1.Test"."Bool"[40]);
   #statTonTime[540].TON(IN := #_w1 AND "Unit1.Em5.ControlNodes".transferPnPLeft."step".transition1[540],
                         PT := #delayTime);
   IF #statTonTime[540].Q THEN
       "Unit1.Em5.ControlNodes".transferPnPLeft.sequence.status.nextStep := #JOB_5_STEP_42;
   END_IF;
END_REGION

REGION Network 43: Step[542] : Transfer PP Left [Unclamp request] => Side Tape Fix Stage
   RUNG wire#powerrail
      { S7_Templates := "SrcType := DInt" } EQ_Contact(in1 := "Unit1.Em5.ControlNodes".transferPnPLeft.sequence.status.currentStep, in2 := #JOB_5_STEP_42)
      Contact( "Unit1.Em5.ControlNodes".transferPnPLeft.sequence.status.seqActive )
      wire#w1
      Coil( "Unit1.Em5.ControlNodes".transferPnPLeft."step".action1[542] )
   END_RUNG
   RUNG wire#w1
      Contact( "Unit1.EmNodes".emRelations.em04.sequence.sideTapeFixStage.jobInterface.unloadJob7.unClampDone )
      wire#w2
      Coil( "Unit1.Em5.ControlNodes".transferPnPLeft."step".transition1[542] )
   END_RUNG
   RUNG wire#w1
      I_Contact( "Unit1.EmNodes".emRelations.em04.isLinked )
   END_RUNG wire#w2
   RUNG wire#w1
      Contact( "Unit1.Em5.ControlNodes".transferPnPLeft."step".transition1[542] )
      { S7_Templates := "time_type := Time" } #statTonTime[542].TON(pt := #delayTime, et =>)
      Move(in := #JOB_5_STEP_80, out1 => "Unit1.Em5.ControlNodes".transferPnPLeft.sequence.status.nextStep)
   END_RUNG
   // the same network as SCL:
   "Unit1.Em5.ControlNodes".transferPnPLeft."step".action1[542] := ("Unit1.Em5.ControlNodes".transferPnPLeft.sequence.status.currentStep = #JOB_5_STEP_42) AND "Unit1.Em5.ControlNodes".transferPnPLeft.sequence.status.seqActive;
   "Unit1.Em5.ControlNodes".transferPnPLeft."step".transition1[542] := ("Unit1.Em5.ControlNodes".transferPnPLeft.sequence.status.currentStep = #JOB_5_STEP_42) AND "Unit1.Em5.ControlNodes".transferPnPLeft.sequence.status.seqActive AND ("Unit1.EmNodes".emRelations.em04.sequence.sideTapeFixStage.jobInterface.unloadJob7.unClampDone OR NOT "Unit1.EmNodes".emRelations.em04.isLinked);
   #statTonTime[542].TON(IN := ("Unit1.Em5.ControlNodes".transferPnPLeft.sequence.status.currentStep = #JOB_5_STEP_42) AND "Unit1.Em5.ControlNodes".transferPnPLeft.sequence.status.seqActive AND "Unit1.Em5.ControlNodes".transferPnPLeft."step".transition1[542],
                         PT := #delayTime);
   IF #statTonTime[542].Q THEN
       "Unit1.Em5.ControlNodes".transferPnPLeft.sequence.status.nextStep := #JOB_5_STEP_80;
   END_IF;
END_REGION

REGION Network 44: Step[580] : Transfer PP Left Y-Axis Wait Pos
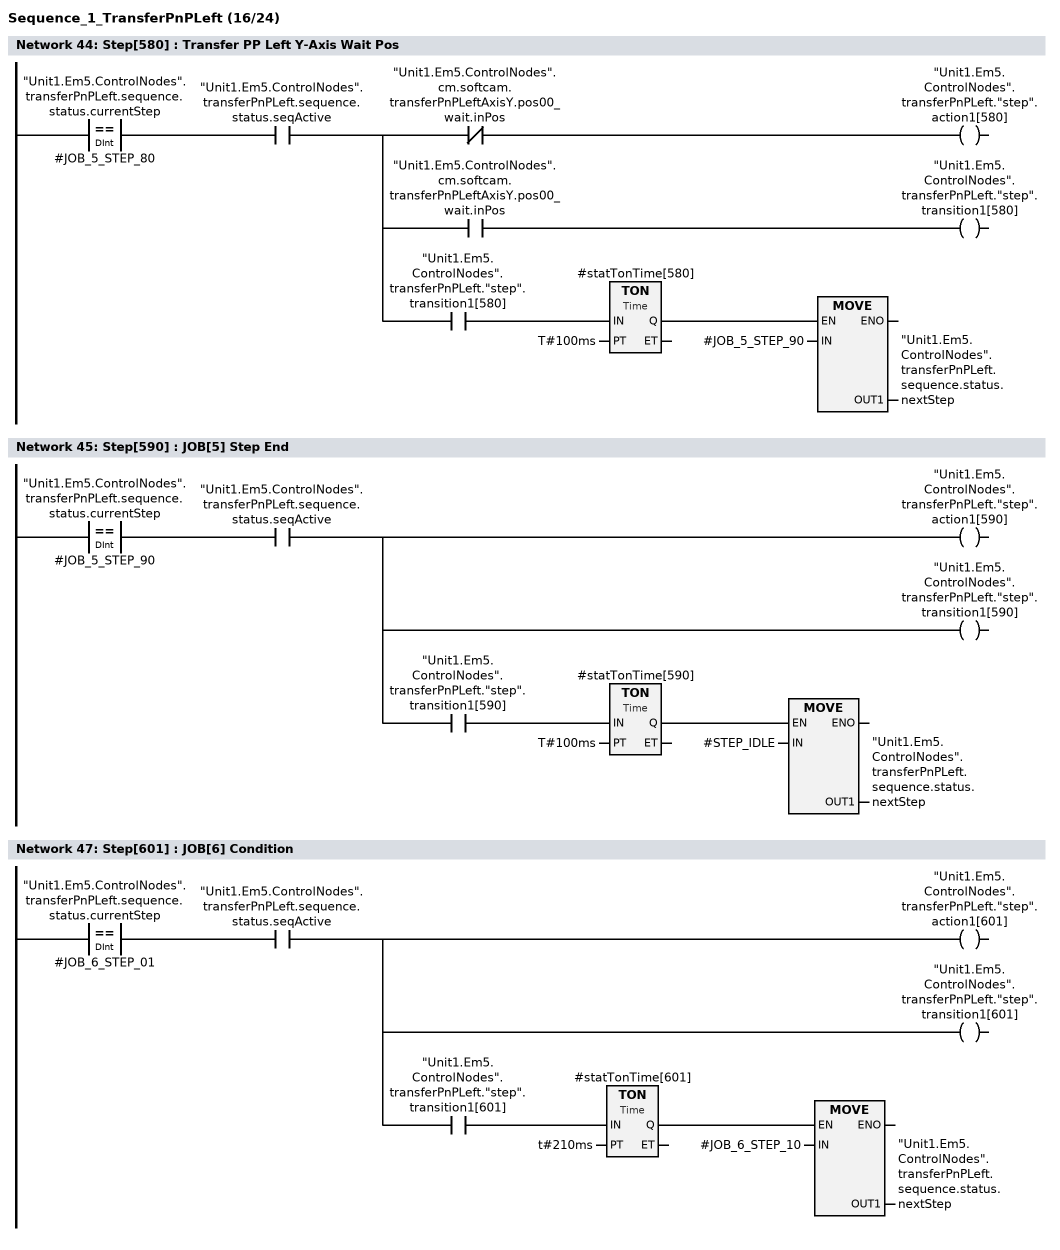
   RUNG wire#powerrail
      { S7_Templates := "SrcType := DInt" } EQ_Contact(in1 := "Unit1.Em5.ControlNodes".transferPnPLeft.sequence.status.currentStep, in2 := #JOB_5_STEP_80)
      Contact( "Unit1.Em5.ControlNodes".transferPnPLeft.sequence.status.seqActive )
      wire#w1
      I_Contact( "Unit1.Em5.ControlNodes".cm.softcam.transferPnPLeftAxisY.pos00_wait.inPos )
      Coil( "Unit1.Em5.ControlNodes".transferPnPLeft."step".action1[580] )
   END_RUNG
   RUNG wire#w1
      Contact( "Unit1.Em5.ControlNodes".cm.softcam.transferPnPLeftAxisY.pos00_wait.inPos )
      Coil( "Unit1.Em5.ControlNodes".transferPnPLeft."step".transition1[580] )
   END_RUNG
   RUNG wire#w1
      Contact( "Unit1.Em5.ControlNodes".transferPnPLeft."step".transition1[580] )
      { S7_Templates := "time_type := Time" } #statTonTime[580].TON(pt := T#100ms, et =>)
      Move(in := #JOB_5_STEP_90, out1 => "Unit1.Em5.ControlNodes".transferPnPLeft.sequence.status.nextStep)
   END_RUNG
   // the same network as SCL:
   #_w1 := ("Unit1.Em5.ControlNodes".transferPnPLeft.sequence.status.currentStep = #JOB_5_STEP_80) AND "Unit1.Em5.ControlNodes".transferPnPLeft.sequence.status.seqActive;
   "Unit1.Em5.ControlNodes".transferPnPLeft."step".action1[580] := #_w1 AND NOT "Unit1.Em5.ControlNodes".cm.softcam.transferPnPLeftAxisY.pos00_wait.inPos;
   "Unit1.Em5.ControlNodes".transferPnPLeft."step".transition1[580] := #_w1 AND "Unit1.Em5.ControlNodes".cm.softcam.transferPnPLeftAxisY.pos00_wait.inPos;
   #statTonTime[580].TON(IN := #_w1 AND "Unit1.Em5.ControlNodes".transferPnPLeft."step".transition1[580],
                         PT := T#100ms);
   IF #statTonTime[580].Q THEN
       "Unit1.Em5.ControlNodes".transferPnPLeft.sequence.status.nextStep := #JOB_5_STEP_90;
   END_IF;
END_REGION

REGION Network 45: Step[590] : JOB[5] Step End
   RUNG wire#powerrail
      { S7_Templates := "SrcType := DInt" } EQ_Contact(in1 := "Unit1.Em5.ControlNodes".transferPnPLeft.sequence.status.currentStep, in2 := #JOB_5_STEP_90)
      Contact( "Unit1.Em5.ControlNodes".transferPnPLeft.sequence.status.seqActive )
      wire#w1
      Coil( "Unit1.Em5.ControlNodes".transferPnPLeft."step".action1[590] )
   END_RUNG
   RUNG wire#w1
      Coil( "Unit1.Em5.ControlNodes".transferPnPLeft."step".transition1[590] )
   END_RUNG
   RUNG wire#w1
      Contact( "Unit1.Em5.ControlNodes".transferPnPLeft."step".transition1[590] )
      { S7_Templates := "time_type := Time" } #statTonTime[590].TON(pt := T#100ms, et =>)
      Move(in := #STEP_IDLE, out1 => "Unit1.Em5.ControlNodes".transferPnPLeft.sequence.status.nextStep)
   END_RUNG
   // the same network as SCL:
   "Unit1.Em5.ControlNodes".transferPnPLeft."step".action1[590] := ("Unit1.Em5.ControlNodes".transferPnPLeft.sequence.status.currentStep = #JOB_5_STEP_90) AND "Unit1.Em5.ControlNodes".transferPnPLeft.sequence.status.seqActive;
   "Unit1.Em5.ControlNodes".transferPnPLeft."step".transition1[590] := ("Unit1.Em5.ControlNodes".transferPnPLeft.sequence.status.currentStep = #JOB_5_STEP_90) AND "Unit1.Em5.ControlNodes".transferPnPLeft.sequence.status.seqActive;
   #statTonTime[590].TON(IN := ("Unit1.Em5.ControlNodes".transferPnPLeft.sequence.status.currentStep = #JOB_5_STEP_90) AND "Unit1.Em5.ControlNodes".transferPnPLeft.sequence.status.seqActive AND "Unit1.Em5.ControlNodes".transferPnPLeft."step".transition1[590],
                         PT := T#100ms);
   IF #statTonTime[590].Q THEN
       "Unit1.Em5.ControlNodes".transferPnPLeft.sequence.status.nextStep := #STEP_IDLE;
   END_IF;
END_REGION

REGION Network 46: *********** JOB[6] HOT PRESS RIGHT JR PUT=AUTO-[B] *************
END_REGION

REGION Network 47: Step[601] : JOB[6] Condition
   RUNG wire#powerrail
      { S7_Templates := "SrcType := DInt" } EQ_Contact(in1 := "Unit1.Em5.ControlNodes".transferPnPLeft.sequence.status.currentStep, in2 := #JOB_6_STEP_01)
      Contact( "Unit1.Em5.ControlNodes".transferPnPLeft.sequence.status.seqActive )
      wire#w1
      Coil( "Unit1.Em5.ControlNodes".transferPnPLeft."step".action1[601] )
   END_RUNG
   RUNG wire#w1
      Coil( "Unit1.Em5.ControlNodes".transferPnPLeft."step".transition1[601] )
   END_RUNG
   RUNG wire#w1
      Contact( "Unit1.Em5.ControlNodes".transferPnPLeft."step".transition1[601] )
      { S7_Templates := "time_type := Time" } #statTonTime[601].TON(pt := t#210ms, et =>)
      Move(in := #JOB_6_STEP_10, out1 => "Unit1.Em5.ControlNodes".transferPnPLeft.sequence.status.nextStep)
   END_RUNG
   // the same network as SCL:
   "Unit1.Em5.ControlNodes".transferPnPLeft."step".action1[601] := ("Unit1.Em5.ControlNodes".transferPnPLeft.sequence.status.currentStep = #JOB_6_STEP_01) AND "Unit1.Em5.ControlNodes".transferPnPLeft.sequence.status.seqActive;
   "Unit1.Em5.ControlNodes".transferPnPLeft."step".transition1[601] := ("Unit1.Em5.ControlNodes".transferPnPLeft.sequence.status.currentStep = #JOB_6_STEP_01) AND "Unit1.Em5.ControlNodes".transferPnPLeft.sequence.status.seqActive;
   #statTonTime[601].TON(IN := ("Unit1.Em5.ControlNodes".transferPnPLeft.sequence.status.currentStep = #JOB_6_STEP_01) AND "Unit1.Em5.ControlNodes".transferPnPLeft.sequence.status.seqActive AND "Unit1.Em5.ControlNodes".transferPnPLeft."step".transition1[601],
                         PT := t#210ms);
   IF #statTonTime[601].Q THEN
       "Unit1.Em5.ControlNodes".transferPnPLeft.sequence.status.nextStep := #JOB_6_STEP_10;
   END_IF;
END_REGION

REGION Network 48: Step[610] : Transfer PP Left X/Z-Axis Hot Press Right Pos
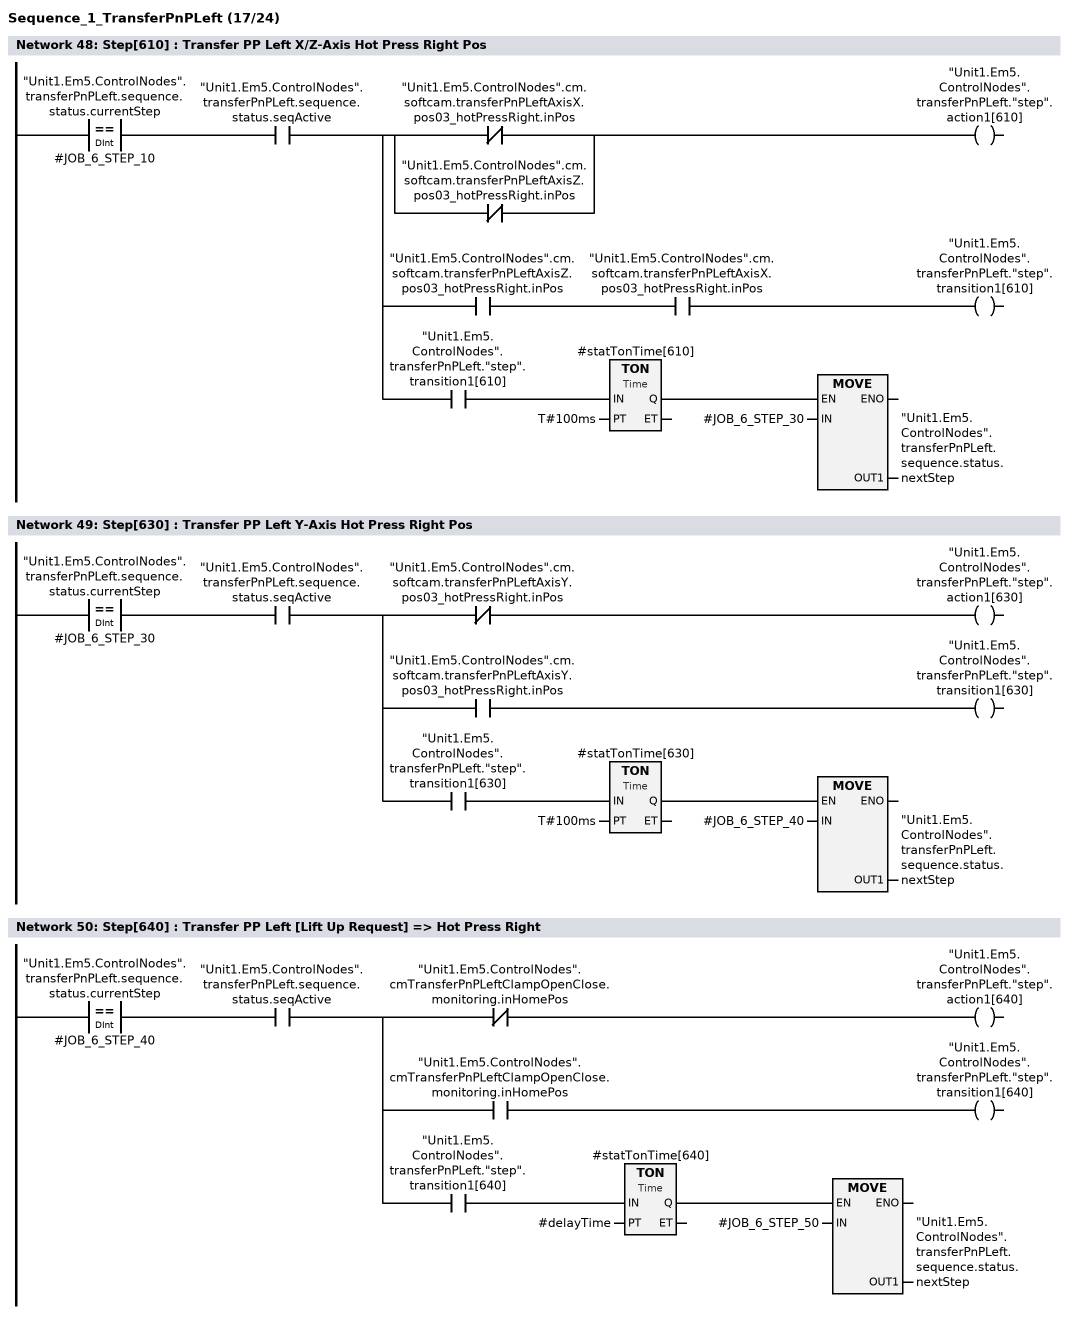
   RUNG wire#powerrail
      { S7_Templates := "SrcType := DInt" } EQ_Contact(in1 := "Unit1.Em5.ControlNodes".transferPnPLeft.sequence.status.currentStep, in2 := #JOB_6_STEP_10)
      Contact( "Unit1.Em5.ControlNodes".transferPnPLeft.sequence.status.seqActive )
      wire#w1
      I_Contact( "Unit1.Em5.ControlNodes".cm.softcam.transferPnPLeftAxisX.pos03_hotPressRight.inPos )
      wire#w2
      Coil( "Unit1.Em5.ControlNodes".transferPnPLeft."step".action1[610] )
   END_RUNG
   RUNG wire#w1
      I_Contact( "Unit1.Em5.ControlNodes".cm.softcam.transferPnPLeftAxisZ.pos03_hotPressRight.inPos )
   END_RUNG wire#w2
   RUNG wire#w1
      Contact( "Unit1.Em5.ControlNodes".cm.softcam.transferPnPLeftAxisZ.pos03_hotPressRight.inPos )
      Contact( "Unit1.Em5.ControlNodes".cm.softcam.transferPnPLeftAxisX.pos03_hotPressRight.inPos )
      Coil( "Unit1.Em5.ControlNodes".transferPnPLeft."step".transition1[610] )
   END_RUNG
   RUNG wire#w1
      Contact( "Unit1.Em5.ControlNodes".transferPnPLeft."step".transition1[610] )
      { S7_Templates := "time_type := Time" } #statTonTime[610].TON(pt := T#100ms, et =>)
      Move(in := #JOB_6_STEP_30, out1 => "Unit1.Em5.ControlNodes".transferPnPLeft.sequence.status.nextStep)
   END_RUNG
   // the same network as SCL:
   #_w1 := ("Unit1.Em5.ControlNodes".transferPnPLeft.sequence.status.currentStep = #JOB_6_STEP_10) AND "Unit1.Em5.ControlNodes".transferPnPLeft.sequence.status.seqActive;
   "Unit1.Em5.ControlNodes".transferPnPLeft."step".action1[610] := #_w1 AND (NOT "Unit1.Em5.ControlNodes".cm.softcam.transferPnPLeftAxisX.pos03_hotPressRight.inPos OR NOT "Unit1.Em5.ControlNodes".cm.softcam.transferPnPLeftAxisZ.pos03_hotPressRight.inPos);
   "Unit1.Em5.ControlNodes".transferPnPLeft."step".transition1[610] := #_w1 AND "Unit1.Em5.ControlNodes".cm.softcam.transferPnPLeftAxisZ.pos03_hotPressRight.inPos AND "Unit1.Em5.ControlNodes".cm.softcam.transferPnPLeftAxisX.pos03_hotPressRight.inPos;
   #statTonTime[610].TON(IN := #_w1 AND "Unit1.Em5.ControlNodes".transferPnPLeft."step".transition1[610],
                         PT := T#100ms);
   IF #statTonTime[610].Q THEN
       "Unit1.Em5.ControlNodes".transferPnPLeft.sequence.status.nextStep := #JOB_6_STEP_30;
   END_IF;
END_REGION

REGION Network 49: Step[630] : Transfer PP Left Y-Axis Hot Press Right Pos
   RUNG wire#powerrail
      { S7_Templates := "SrcType := DInt" } EQ_Contact(in1 := "Unit1.Em5.ControlNodes".transferPnPLeft.sequence.status.currentStep, in2 := #JOB_6_STEP_30)
      Contact( "Unit1.Em5.ControlNodes".transferPnPLeft.sequence.status.seqActive )
      wire#w1
      I_Contact( "Unit1.Em5.ControlNodes".cm.softcam.transferPnPLeftAxisY.pos03_hotPressRight.inPos )
      Coil( "Unit1.Em5.ControlNodes".transferPnPLeft."step".action1[630] )
   END_RUNG
   RUNG wire#w1
      Contact( "Unit1.Em5.ControlNodes".cm.softcam.transferPnPLeftAxisY.pos03_hotPressRight.inPos )
      Coil( "Unit1.Em5.ControlNodes".transferPnPLeft."step".transition1[630] )
   END_RUNG
   RUNG wire#w1
      Contact( "Unit1.Em5.ControlNodes".transferPnPLeft."step".transition1[630] )
      { S7_Templates := "time_type := Time" } #statTonTime[630].TON(pt := T#100ms, et =>)
      Move(in := #JOB_6_STEP_40, out1 => "Unit1.Em5.ControlNodes".transferPnPLeft.sequence.status.nextStep)
   END_RUNG
   // the same network as SCL:
   #_w1 := ("Unit1.Em5.ControlNodes".transferPnPLeft.sequence.status.currentStep = #JOB_6_STEP_30) AND "Unit1.Em5.ControlNodes".transferPnPLeft.sequence.status.seqActive;
   "Unit1.Em5.ControlNodes".transferPnPLeft."step".action1[630] := #_w1 AND NOT "Unit1.Em5.ControlNodes".cm.softcam.transferPnPLeftAxisY.pos03_hotPressRight.inPos;
   "Unit1.Em5.ControlNodes".transferPnPLeft."step".transition1[630] := #_w1 AND "Unit1.Em5.ControlNodes".cm.softcam.transferPnPLeftAxisY.pos03_hotPressRight.inPos;
   #statTonTime[630].TON(IN := #_w1 AND "Unit1.Em5.ControlNodes".transferPnPLeft."step".transition1[630],
                         PT := T#100ms);
   IF #statTonTime[630].Q THEN
       "Unit1.Em5.ControlNodes".transferPnPLeft.sequence.status.nextStep := #JOB_6_STEP_40;
   END_IF;
END_REGION

REGION Network 50: Step[640] : Transfer PP Left [Lift Up Request] => Hot Press Right
   RUNG wire#powerrail
      { S7_Templates := "SrcType := DInt" } EQ_Contact(in1 := "Unit1.Em5.ControlNodes".transferPnPLeft.sequence.status.currentStep, in2 := #JOB_6_STEP_40)
      Contact( "Unit1.Em5.ControlNodes".transferPnPLeft.sequence.status.seqActive )
      wire#w1
      I_Contact( "Unit1.Em5.ControlNodes".cmTransferPnPLeftClampOpenClose.monitoring.inHomePos )
      Coil( "Unit1.Em5.ControlNodes".transferPnPLeft."step".action1[640] )
   END_RUNG
   RUNG wire#w1
      Contact( "Unit1.Em5.ControlNodes".cmTransferPnPLeftClampOpenClose.monitoring.inHomePos )
      Coil( "Unit1.Em5.ControlNodes".transferPnPLeft."step".transition1[640] )
   END_RUNG
   RUNG wire#w1
      Contact( "Unit1.Em5.ControlNodes".transferPnPLeft."step".transition1[640] )
      { S7_Templates := "time_type := Time" } #statTonTime[640].TON(pt := #delayTime, et =>)
      Move(in := #JOB_6_STEP_50, out1 => "Unit1.Em5.ControlNodes".transferPnPLeft.sequence.status.nextStep)
   END_RUNG
   // the same network as SCL:
   #_w1 := ("Unit1.Em5.ControlNodes".transferPnPLeft.sequence.status.currentStep = #JOB_6_STEP_40) AND "Unit1.Em5.ControlNodes".transferPnPLeft.sequence.status.seqActive;
   "Unit1.Em5.ControlNodes".transferPnPLeft."step".action1[640] := #_w1 AND NOT "Unit1.Em5.ControlNodes".cmTransferPnPLeftClampOpenClose.monitoring.inHomePos;
   "Unit1.Em5.ControlNodes".transferPnPLeft."step".transition1[640] := #_w1 AND "Unit1.Em5.ControlNodes".cmTransferPnPLeftClampOpenClose.monitoring.inHomePos;
   #statTonTime[640].TON(IN := #_w1 AND "Unit1.Em5.ControlNodes".transferPnPLeft."step".transition1[640],
                         PT := #delayTime);
   IF #statTonTime[640].Q THEN
       "Unit1.Em5.ControlNodes".transferPnPLeft.sequence.status.nextStep := #JOB_6_STEP_50;
   END_IF;
END_REGION

